# B&R Automation Studio project Panasonic_LinkaPowerCP2_A2021055 (part 18)

#### Main.st - Init, cyclic, exit code
```iecst
PROGRAM _INIT
	(* Insert code here *)

END_PROGRAM

PROGRAM _CYCLIC

    //Volanie funkcie SequenceControl//
	SequenceControl(SC:= SC_P2_StoperMaticovacky);

	//Volanie podprogramov//
	OvlCentrovacky;
	IOLinkKomunikacia;
	AtlasCopcoKomunikacia;

	//Reset sekcie //
	IF P2_StoperMaticovacky.Reset THEN
		SC_P2_StoperMaticovacky.Step:= 0;
		P2_StoperMaticovacky.Reset:= FALSE;
	ELSIF NOT Safety.STAV.Linka_ZonaCS_AKTIVNA AND NOT P2_StoperMaticovacky.Automat THEN
		SC_P2_StoperMaticovacky.Step:= 0;
	ELSIF NOT Safety.STAV.Linka_ZonaCS_AKTIVNA AND P2_StoperMaticovacky.Automat THEN
		P2_Pracovisko.STAV.Porucha_ST2:= TRUE;
	END_IF

	//Zrušenie podania matice//
	IF P2_StoperMaticovacky.SkrutSet_MaticaM4.CMD.PodajMaticu AND P2_StoperMaticovacky.SkrutSet_MaticaM4.STAV.MaticaPripravena THEN
		P2_StoperMaticovacky.SkrutSet_MaticaM4.CMD.PodajMaticu:= FALSE;
	ELSIF P2_StoperMaticovacky.SkrutSet_MaticaM4.CMD.PodajMaticu AND P2_StoperMaticovacky.SkrutSet_MaticaM4.STAV.ERROR THEN
		P2_StoperMaticovacky.SkrutSet_MaticaM4.CMD.PodajMaticu:= FALSE;
		P2_Alarmy[298]:= TRUE;
		P2_Pracovisko.STAV.Porucha_ST2:= TRUE;
	END_IF

	//Ukončenie komunikácie pri poruche//
	IF P2_Pracovisko.STAV.Porucha_ST2 AND NOT Triger_0 THEN
		Triger_0:= TRUE;
		IF P2_StoperMaticovacky.STAV.VyrobaZacala THEN
			Paletka[i].PAR.StavPowerCP:= 'FAIL';
			Paletka[i].STAV.StavPaletky:= 'NG';
			P2_StoperMaticovacky.KoniecCyklu:= TRUE;
			SC_P2_StoperMaticovacky.ResetStep:= TRUE;
			SC_P2_StoperMaticovacky.Step:= 550;
		ELSE
			SC_P2_StoperMaticovacky.ResetStep:= TRUE;
			SC_P2_StoperMaticovacky.Step:= 0;
		END_IF
	END_IF

	IF NOT P2_Pracovisko.STAV.Porucha_ST2 THEN
		Triger_0:= FALSE;
	END_IF

	CASE SC_P2_StoperMaticovacky.Step OF

		0:
			SC_P2_StoperMaticovacky.StepName:='0 - Nulovanie';
			SC_OvlCentrovacky.Step:= 0;
			P2_StoperMaticovacky.Automat:= FALSE;
			P2_StoperMaticovacky.KoniecCyklu:= FALSE;
			P2_StoperMaticovacky.Manual:= FALSE;
			P2_StoperMaticovacky.STAV.PoINIT:= FALSE;
			P2_StoperMaticovacky.STAV.VyrobaZacala:= FALSE;
			P2_StoperMaticovacky.STAV.VstupnaKamerovaKontrola:= FALSE;
			P2_StoperMaticovacky.OUT.ZasunStoper:= FALSE;
			P2_StoperMaticovacky.OUT.Maticovacku_M4_VYSUN:= FALSE;
			P2_StoperMaticovacky.OUT.Maticovacka_M4_Odvzdusn_ON:= FALSE;
			P2_StoperMaticovacky.OUT.Maticovacka_M4_Prisavanie_ON:= FALSE;
			P2_StoperMaticovacky.RFID_hlava.PrecitajChipRFID:= FALSE;
			P2_StoperMaticovacky.SkrutSet_MaticaM4.CMD.ENABLE:= FALSE;

			P2_StoperMaticovacky.Maticovacka_M4.RESET_Poruchy:= FALSE;
			P2_StoperMaticovacky.Maticovacka_M4.RESET_Vysledkov:= FALSE;
			P2_StoperMaticovacky.Maticovacka_M4.START_Skrutkovania:= FALSE;
			P2_StoperMaticovacky.Maticovacka_M4.START_Utahovania:= FALSE;
			P2_StoperMaticovacky.CMD.RR_VysunCentrovanie:= FALSE;

			CAM9.CMD.Triger:= FALSE;
			CAM9.STAV.Results_READY:= FALSE;
			FTP_CAM9.CMD.OdosliFotku:= FALSE;
			FTP_CAM9.CMD.VymazFotku:= FALSE;
			TRCB_P2_Maticovacka_ST4.CMD.VyziadajStavPaletky_TYP1:= FALSE;
			TRCB_P2_Maticovacka_ST4.CMD.PriradQRkodFiltra_TYP3:= FALSE;
			TRCB_P2_Maticovacka_ST4.CMD.OdosliStavPaletky_TYP2:= FALSE;
			TRCB_P2_Maticovacka_ST4.CMD.VyziadajStavPanatrace_TYP4:= FALSE;

			P2_StoperMaticovacky.STAV.PrebiehaVyvezeniePaletky:= FALSE;
			P2_StoperZaklTesnenia.STAV.PrebiehaVyvezeniePaletky:= FALSE;
			P2_Maticov_KAM_Result_Ignoruj:= FALSE;
			TestovaciKus:= FALSE;
			CisloFotky:= 0;
			P2_Maticov_KAM_Result_OK:= FALSE;
			P2_Maticov_KAM_Result_NG:= FALSE;
			P2_Vizu.ZobrazHL1_ST4:= FALSE;
			P2_Vizu.ZobrazHL2_ST4:= FALSE;
			P2_Vizu.ZobrazHL3_ST4:= FALSE;
			P2_Vizu.ZobrazHL4_ST4:= FALSE;
			TRCB_P2_Maticov_OpatovnyDopyt:= FALSE;
			TRCB_P2_Maticov_PaletkaNG:= FALSE;
			VysunutieSkrutkovacky_OK:= FALSE;
			PocetTrigrovKamery:= 0;
			PocetDopytovNaServer:= 0;
			CasSrobovania:= 0;
			P2_Maticovacka_Taktime.IN.START_MeraniaCasu:= FALSE;
			P2_Maticovacka_Taktime.IN.START_MeraniaStratovehoCasu:= FALSE;

			IF Safety.STAV.Linka_ZonaCS_AKTIVNA AND
				Safety.STAV.P2_ZonaBunky_AKTIVNA AND
				P2_Pracovisko.STAV.HardwareBunky_OK AND
				NOT P2_Pracovisko.STAV.Porucha_ST2 AND
				NOT P2_Pracovisko.STAV.Porucha_ST3 AND
				NOT P2_Pracovisko.STAV.Porucha_ST4 AND
				NOT P2_Pracovisko.STAV.Porucha_ST5 THEN
				SC_P2_StoperMaticovacky.ResetStep:= TRUE;
				SC_P2_StoperMaticovacky.Step:= 1;
			END_IF

		1:
			SC_P2_StoperMaticovacky.StepName:='1 - Cakam na spustenie vyroby';
			P2_StoperMaticovacky.KoniecCyklu:= FALSE;
			IF P2_StoperMaticovacky.Automat THEN
				SC_P2_StoperMaticovacky.Step:= 2;
			ELSIF P2_StoperMaticovacky.Manual THEN
				SC_P2_StoperMaticovacky.Step:= 700;
			END_IF

			//********************************************************Inicializácia****************************************************************************//

		2:
			SC_P2_StoperMaticovacky.StepName:='2 - Inicializacia - cakam na spustenie inicializacie';
			SC_P2_StoperMaticovacky.IdleTime.PT:= T#4s;
			SC_P2_StoperMaticovacky.AlarmTime.PT:= T#5s;

			P2_StoperMaticovacky.OUT.Maticovacku_M4_VYSUN:= FALSE;

			IF P2_StoperMaticovacky.IN.Maticovacka_M4_ZASUNUTA AND P2_Dopravniky.STAV.PoINIT THEN
				P2_StoperMaticovacky.SkrutSet_MaticaM4.CMD.ENABLE:= TRUE;
				SC_P2_StoperMaticovacky.ResetStep:= TRUE;
				SC_P2_StoperMaticovacky.Step:= 10;
			END_IF

		3:
			SC_P2_StoperMaticovacky.StepName:='3 - Inicializacia - vymazanie adresara kamery';
			SC_P2_StoperMaticovacky.IdleTime.PT:= T#4s;
			SC_P2_StoperMaticovacky.AlarmTime.PT:= T#5s;

			IF NOT SC_P2_StoperMaticovacky.Switch1 THEN
				FTP_CAM9.CMD.VymazFotku:= TRUE;
				SC_P2_StoperMaticovacky.Switch1:= TRUE;
			END_IF

			IF FTP_CAM9.STATUS.KomunikaciaUkoncena THEN
				FTP_CAM9.CMD.VymazFotku:= FALSE;
				SC_P2_StoperMaticovacky.ResetStep:= TRUE;
				SC_P2_StoperMaticovacky.Step:= 10;
			ELSIF FTP_CAM9.STATUS.KomunikaciaError THEN
				P2_Alarmy[229]:= TRUE;
				P2_Pracovisko.STAV.Porucha_ST2:= TRUE;
			END_IF

		10:
			SC_P2_StoperMaticovacky.StepName:='10 - Inicializacia - zasunutie centrovacky';
			SC_P2_StoperMaticovacky.IdleTime.PT:= T#4s;
			SC_P2_StoperMaticovacky.AlarmTime.PT:= T#5s;

			IF NOT SC_P2_StoperMaticovacky.Switch1 THEN
				Centrovacku_ZASUN:= TRUE;
				SC_P2_StoperMaticovacky.Switch1:= TRUE;
			END_IF

			IF P2_StoperMaticovacky.IN.Centrovanie_ZASUNUTE AND P2_Dopravniky.STAV.PoINIT THEN
				SC_P2_StoperMaticovacky.ResetStep:= TRUE;
				SC_P2_StoperMaticovacky.Step:= 12;
			END_IF

		12:
			SC_P2_StoperMaticovacky.StepName:='12 - Inicializacia - kontrola matice v maticovacke';
			SC_P2_StoperMaticovacky.IdleTime.PT:= T#5s;
			SC_P2_StoperMaticovacky.AlarmTime.PT:= T#10s;

			IF NOT SC_P2_StoperMaticovacky.Switch1 AND NOT P2_StoperMaticovacky.SkrutSet_MaticaM4.STAV.MaticaPripravena THEN
				P2_StoperMaticovacky.SkrutSet_MaticaM4.CMD.PodajMaticu:= TRUE;
				SC_P2_StoperMaticovacky.Switch1:= TRUE;
			END_IF

			IF P2_StoperMaticovacky.SkrutSet_MaticaM4.STAV.MaticaPripravena THEN
				SC_P2_StoperMaticovacky.ResetStep:= TRUE;
				SC_P2_StoperMaticovacky.Step:= 13;
			END_IF

		13:
			SC_P2_StoperMaticovacky.StepName:='13 - Inicializacia - hladanie paletky';
			SC_P2_StoperMaticovacky.IdleTime.PT:= T#5s;
			SC_P2_StoperMaticovacky.AlarmTime.PT:= T#5s;
			SC_P2_StoperMaticovacky.IdleTime.IN:= TRUE;

			IF P2_StoperMaticovacky.RFID_hlava.PritomnostPaletky THEN
				SC_P2_StoperMaticovacky.ResetStep:= TRUE;
				SC_P2_StoperMaticovacky.Step:= 20;
			ELSIF SC_P2_StoperMaticovacky.IdleTime.Q THEN
				P2_StoperMaticovacky.STAV.PoINIT:= TRUE;
				SC_P2_StoperMaticovacky.ResetStep:= TRUE;
				SC_P2_StoperMaticovacky.Step:= 100;
			END_IF

		20:
			SC_P2_StoperMaticovacky.StepName:='20 - Inicializacia - precitanie cisla paletky';
			SC_P2_StoperMaticovacky.IdleTime.PT:= T#200ms;
			SC_P2_StoperMaticovacky.AlarmTime.PT:= T#5s;

			SC_P2_StoperMaticovacky.IdleTime.IN:= P2_StoperMaticovacky.RFID_hlava.PritomnostPaletky;

			IF SC_P2_StoperMaticovacky.IdleTime.Q AND NOT SC_P2_StoperMaticovacky.Switch1 THEN
				P2_StoperMaticovacky.RFID_hlava.PrecitajChipRFID:= TRUE;
				i:= 0;
				SC_P2_StoperMaticovacky.Switch1:= TRUE;
			END_IF

			IF P2_StoperMaticovacky.RFID_hlava.Stav_CitanieZapis_OK AND P2_StoperMaticovacky.RFID_hlava.PrecitaneCisloPaletky <> 0 THEN
				i:= P2_StoperMaticovacky.RFID_hlava.PrecitaneCisloPaletky;
				P2_StoperMaticovacky.PAR.CisloPaletky:= P2_StoperMaticovacky.RFID_hlava.PrecitaneCisloPaletky;
				P2_StoperMaticovacky.RFID_hlava.PrecitajChipRFID:= FALSE;
				SC_P2_StoperMaticovacky.ResetStep:= TRUE;
				SC_P2_StoperMaticovacky.Step:= 23;
			END_IF

		23:
			SC_P2_StoperMaticovacky.StepName:='23 - Inicializacia - kontrola a priradenie indexu paletky na zaklade precitanej hodnoty';
			SC_P2_StoperMaticovacky.IdleTime.PT:= T#1s;
			SC_P2_StoperMaticovacky.AlarmTime.PT:= T#5s;

			IF i<> 0 THEN
				P2_StoperMaticovacky.PAR.CisloPaletky_STRING:= USINT_TO_STRING(i);
				Paletka[i].PAR.CisloPaletky:= USINT_TO_STRING(i);
				SC_P2_StoperMaticovacky.ResetStep:= TRUE;
				SC_P2_StoperMaticovacky.Step:= 30;
			ELSE
				P2_Alarmy[211]:= TRUE;
				P2_Pracovisko.STAV.Porucha_ST2:= TRUE;
			END_IF

		30:
			SC_P2_StoperMaticovacky.StepName:='30 - Inicializacia - kontrola stavu paletky';
			SC_P2_StoperMaticovacky.IdleTime.PT:= T#200ms;
			SC_P2_StoperMaticovacky.AlarmTime.PT:= T#5s;

			IF Paletka[i].STAV.StavPaletky = '' THEN
				Paletka[i].STAV.StavPaletky:= 'NG';
				SC_P2_StoperMaticovacky.ResetStep:= TRUE;
				SC_P2_StoperMaticovacky.Step:= 560;
			ELSIF Paletka[i].STAV.StavPaletky = 'PRECH' THEN
				P2_StoperMaticovacky.STAV.PoINIT:= TRUE;
				SC_P2_StoperMaticovacky.ResetStep:= TRUE;
				SC_P2_StoperMaticovacky.Step:= 560;
			ELSIF Paletka[i].STAV.StavPaletky = 'TEST' AND Paletka[i].STAV.CisloTestovacejStanice = 'ST_4' THEN
				TestovaciKus:= TRUE;
			ELSIF Paletka[i].STAV.StavPaletky = 'TEST' AND Paletka[i].STAV.CisloTestovacejStanice <> 'ST_4' THEN
				P2_StoperMaticovacky.STAV.PoINIT:= TRUE;
				SC_P2_StoperMaticovacky.ResetStep:= TRUE;
				SC_P2_StoperMaticovacky.Step:= 560;
			ELSIF Paletka[i].STAV.StavPaletky = 'REV' AND Paletka[i].STAV.CisloRevorkovejStanice = 'ST_4' THEN
				Paletka[i].STAV.StavPaletky:= 'OK';
				SC_P2_StoperMaticovacky.ResetStep:= TRUE;
				SC_P2_StoperMaticovacky.Step:= 33;
			ELSIF Paletka[i].STAV.StavPaletky = 'REV' AND Paletka[i].STAV.CisloRevorkovejStanice <> 'ST_4' THEN
				P2_StoperMaticovacky.STAV.PoINIT:= TRUE;
				SC_P2_StoperMaticovacky.ResetStep:= TRUE;
				SC_P2_StoperMaticovacky.Step:= 560;
			ELSIF Paletka[i].STAV.StavPaletky = 'OK' THEN
				SC_P2_StoperMaticovacky.ResetStep:= TRUE;
				SC_P2_StoperMaticovacky.Step:= 33;
			ELSIF Paletka[i].STAV.StavPaletky = 'NG' THEN
				P2_StoperMaticovacky.STAV.PoINIT:= TRUE;
				SC_P2_StoperMaticovacky.ResetStep:= TRUE;
				SC_P2_StoperMaticovacky.Step:= 560;
			END_IF

		33:
			SC_P2_StoperMaticovacky.StepName:='33 - Inicializacia - rozhodnutie podla typu modelu';
			SC_P2_StoperMaticovacky.IdleTime.PT:= T#200ms;
			SC_P2_StoperMaticovacky.AlarmTime.PT:= T#5s;

			IF Linka.PAR.ZvolenyModel = '5H' THEN
				SC_P2_StoperMaticovacky.ResetStep:= TRUE;
				SC_P2_StoperMaticovacky.Step:= 35;
			ELSE
				P2_StoperMaticovacky.STAV.PoINIT:= TRUE;
				SC_P2_StoperMaticovacky.ResetStep:= TRUE;
				SC_P2_StoperMaticovacky.Step:= 560;
			END_IF

		35:
			SC_P2_StoperMaticovacky.StepName:='35 - Inicializacia - kontrola uzavretia komunikacie';
			SC_P2_StoperMaticovacky.IdleTime.PT:= T#200ms;
			SC_P2_StoperMaticovacky.AlarmTime.PT:= T#5s;

			IF Paletka[i].STAV.Komunikacia_DONE THEN
				P2_StoperMaticovacky.STAV.PoINIT:= TRUE;
				SC_P2_StoperMaticovacky.ResetStep:= TRUE;
				SC_P2_StoperMaticovacky.Step:= 560;
			ELSE
				P2_StoperMaticovacky.STAV.PoINIT:= TRUE;
				P2_StoperMaticovacky.STAV.VstupnaKamerovaKontrola:= TRUE;
				SC_P2_StoperMaticovacky.ResetStep:= TRUE;
				SC_P2_StoperMaticovacky.Step:= 100;
			END_IF

			//********************************************************Automatický režim****************************************************************************//

		100:
			SC_P2_StoperMaticovacky.StepName:='100 - Automaticky Rezim - cakam na príchod paletky na stoper';
			SC_P2_StoperMaticovacky.IdleTime.PT:= T#200ms;
			SC_P2_StoperMaticovacky.AlarmTime.PT:= T#5s;

			SC_P2_StoperMaticovacky.IdleTime.IN:= P2_StoperMaticovacky.RFID_hlava.PritomnostPaletky;

			IF P2_StoperMaticovacky.RFID_hlava.PritomnostPaletky THEN
				P2_StoperZaklTesnenia.STAV.PrebiehaVyvezeniePaletky:= FALSE;
			END_IF

			IF NOT SC_P2_StoperMaticovacky.Switch1 AND P2_StoperMaticovacky.RFID_hlava.PritomnostPaletky THEN
				P2_Maticovacka_Taktime.IN.START_MeraniaCasu:= TRUE;
				P2_Maticovacka_Taktime.IN.ZAPIS_MeraniaCasu:= TRUE;
				P2_Maticovacka_Taktime.IN.ZAPIS_StratovyCas:= TRUE;
				Buffer_4.Hodnota:= P2_Maticovacka_Taktime.OUT.StratoveSekundy;
				Buffer_4.ZapisHodnotu:= TRUE;
				SC_P2_StoperMaticovacky.Switch1:= TRUE;
			END_IF

			IF P2_StoperMaticovacky.KoniecCyklu THEN
				SC_P2_StoperMaticovacky.ResetStep:= TRUE;
				SC_P2_StoperMaticovacky.Step:= 0;
			ELSIF SC_P2_StoperMaticovacky.IdleTime.Q THEN
				SC_P2_StoperMaticovacky.ResetStep:= TRUE;
				SC_P2_StoperMaticovacky.Step:= 101;
			END_IF

		101:
			SC_P2_StoperMaticovacky.StepName:='101 - Automaticky Rezim - precitanie cisla paletky';
			SC_P2_StoperMaticovacky.IdleTime.PT:= T#500ms;
			SC_P2_StoperMaticovacky.AlarmTime.PT:= T#5s;
			SC_P2_StoperMaticovacky.IdleTime.IN:= TRUE;

			IF NOT SC_P2_StoperMaticovacky.Switch1 THEN
				P2_StoperMaticovacky.RFID_hlava.PrecitajChipRFID:= TRUE;
				i:= 0;
				SC_P2_StoperMaticovacky.Switch1:= TRUE;
			END_IF

			IF P2_StoperMaticovacky.RFID_hlava.Stav_CitanieZapis_OK AND P2_StoperMaticovacky.RFID_hlava.PrecitaneCisloPaletky <> 0 THEN
				i:= P2_StoperMaticovacky.RFID_hlava.PrecitaneCisloPaletky;
				P2_StoperMaticovacky.PAR.CisloPaletky:= P2_StoperMaticovacky.RFID_hlava.PrecitaneCisloPaletky;
				P2_StoperMaticovacky.RFID_hlava.PrecitajChipRFID:= FALSE;
				SC_P2_StoperMaticovacky.ResetStep:= TRUE;
				SC_P2_StoperMaticovacky.Step:= 102;
			END_IF

		102:
			SC_P2_StoperMaticovacky.StepName:='102 - Automaticky Rezim - kontrola a priradenie indexu paletky na zaklade precitanej hodnoty';
			SC_P2_StoperMaticovacky.IdleTime.PT:= T#1s;
			SC_P2_StoperMaticovacky.AlarmTime.PT:= T#5s;

			IF i<> 0 THEN
				P2_StoperMaticovacky.PAR.CisloPaletky_STRING:= USINT_TO_STRING(i);
				Paletka[i].PAR.CisloPaletky:= USINT_TO_STRING(i);
				SC_P2_StoperMaticovacky.ResetStep:= TRUE;
				SC_P2_StoperMaticovacky.Step:= 103;
			ELSE
				P2_Alarmy[211]:= TRUE;
				P2_Pracovisko.STAV.Porucha_ST2:= TRUE;
			END_IF

		103:
			SC_P2_StoperMaticovacky.StepName:='103 - Automaticky Rezim - kontrola stavu paletky';
			SC_P2_StoperMaticovacky.IdleTime.PT:= T#200ms;
			SC_P2_StoperMaticovacky.AlarmTime.PT:= T#5s;

			IF Paletka[i].STAV.StavPaletky = '' THEN
				Paletka[i].STAV.StavPaletky:= 'NG';
				SC_P2_StoperMaticovacky.ResetStep:= TRUE;
				SC_P2_StoperMaticovacky.Step:= 560;
			ELSIF Paletka[i].STAV.StavPaletky = 'PRECH' THEN
				SC_P2_StoperMaticovacky.ResetStep:= TRUE;
				SC_P2_StoperMaticovacky.Step:= 560;
			ELSIF Paletka[i].STAV.StavPaletky = 'TEST' AND Paletka[i].STAV.CisloTestovacejStanice = 'ST_4' THEN
				TestovaciKus:= TRUE;
			ELSIF Paletka[i].STAV.StavPaletky = 'TEST' AND Paletka[i].STAV.CisloTestovacejStanice <> 'ST_4' THEN
				SC_P2_StoperMaticovacky.ResetStep:= TRUE;
				SC_P2_StoperMaticovacky.Step:= 560;
			ELSIF Paletka[i].STAV.StavPaletky = 'REV' AND Paletka[i].STAV.CisloRevorkovejStanice = 'ST_4' THEN
				Paletka[i].STAV.StavPaletky:= 'OK';
				SC_P2_StoperMaticovacky.ResetStep:= TRUE;
				SC_P2_StoperMaticovacky.Step:= 108;
			ELSIF Paletka[i].STAV.StavPaletky = 'REV' AND Paletka[i].STAV.CisloRevorkovejStanice <> 'ST_4' THEN
				SC_P2_StoperMaticovacky.ResetStep:= TRUE;
				SC_P2_StoperMaticovacky.Step:= 560;
			ELSIF Paletka[i].STAV.StavPaletky = 'OK' THEN
				SC_P2_StoperMaticovacky.ResetStep:= TRUE;
				SC_P2_StoperMaticovacky.Step:= 108;
			ELSIF Paletka[i].STAV.StavPaletky = 'NG' THEN
				SC_P2_StoperMaticovacky.ResetStep:= TRUE;
				SC_P2_StoperMaticovacky.Step:= 560;
			END_IF

		108:
			SC_P2_StoperMaticovacky.StepName:='108 - Automaticky Rezim - rozhodnutie podla typu modelu';
			SC_P2_StoperMaticovacky.IdleTime.PT:= T#200ms;
			SC_P2_StoperMaticovacky.AlarmTime.PT:= T#5s;

			IF Linka.PAR.ZvolenyModel = '5H' THEN
				SC_P2_StoperMaticovacky.ResetStep:= TRUE;
				SC_P2_StoperMaticovacky.Step:= 110;
			ELSE
				SC_P2_StoperMaticovacky.ResetStep:= TRUE;   //Paletka iba prechádza
				SC_P2_StoperMaticovacky.Step:= 560;
			END_IF

		110:
			SC_P2_StoperMaticovacky.StepName:='110 - Automaticky Rezim - vyziadanie stavu komunikacie zo serverom';
			SC_P2_StoperMaticovacky.IdleTime.PT:= T#200ms;
			SC_P2_StoperMaticovacky.AlarmTime.PT:= T#10s;

			IF Linka.KOM_Panatrace_OFF THEN
				SC_P2_StoperMaticovacky.ResetStep:= TRUE;
				SC_P2_StoperMaticovacky.Step:= 118;
			ELSIF NOT SC_P2_StoperMaticovacky.Switch1 AND TRCB_P2_Maticovacka_ST4.STATUS.KOM_READY THEN
				TRCB_P2_Maticovacka_ST4.CMD.VyziadajStavPanatrace_TYP4:= TRUE;
				(*P2_Maticovacka_Taktime.IN.START_MeraniaStratovehoCasu:= TRUE;*)
				Centrovacku_VYSUN:= TRUE;
				SC_P2_StoperMaticovacky.Switch1:= TRUE;
			END_IF

			IF TRCB_P2_Maticovacka_ST4.STATUS.KomunikaciaUkoncena THEN
				TRCB_P2_Maticovacka_ST4.CMD.VyziadajStavPanatrace_TYP4:= FALSE;
				P2_Maticovacka_Taktime.IN.START_MeraniaStratovehoCasu:= FALSE;
				SC_P2_StoperMaticovacky.ResetStep:= TRUE;
				SC_P2_StoperMaticovacky.Step:= 111;
			ELSIF TRCB_P2_Maticovacka_ST4.STATUS.KomunikaciaError THEN
				TRCB_P2_Maticovacka_ST4.CMD.VyziadajStavPanatrace_TYP4:= FALSE;
				P2_Maticovacka_Taktime.IN.START_MeraniaStratovehoCasu:= FALSE;
				SC_P2_StoperMaticovacky.ResetStep:= TRUE;
				SC_P2_StoperMaticovacky.Step:= 112;
			END_IF

		111:
			SC_P2_StoperMaticovacky.StepName:='111 - Automaticky Rezim - kontrola odpovede servera';
			SC_P2_StoperMaticovacky.IdleTime.PT:= T#200ms;
			SC_P2_StoperMaticovacky.AlarmTime.PT:= T#5s;

			IF NOT TRCB_P2_Maticovacka_ST4.STATUS.KomunikaciaUkoncena THEN
				IF TRCB_P2_Maticovacka_ST4.OUTPUTS.DruhCinnostiNaPaletke = '0;Generating' THEN
					SC_P2_StoperMaticovacky.ResetStep:= TRUE;
					SC_P2_StoperMaticovacky.Step:= 112;
				ELSIF TRCB_P2_Maticovacka_ST4.OUTPUTS.DruhCinnostiNaPaletke = '1;Request' THEN
					SC_P2_StoperMaticovacky.ResetStep:= TRUE;
					SC_P2_StoperMaticovacky.Step:= 113;
				ELSIF TRCB_P2_Maticovacka_ST4.OUTPUTS.DruhCinnostiNaPaletke = '2;Report' THEN
					SC_P2_StoperMaticovacky.ResetStep:= TRUE;
					SC_P2_StoperMaticovacky.Step:= 118;
				ELSIF TRCB_P2_Maticovacka_ST4.OUTPUTS.DruhCinnostiNaPaletke = '3;Wedding' THEN
					SC_P2_StoperMaticovacky.ResetStep:= TRUE;
					SC_P2_StoperMaticovacky.Step:= 112;
				ELSIF TRCB_P2_Maticovacka_ST4.OUTPUTS.DruhCinnostiNaPaletke = '4;Status' THEN
					SC_P2_StoperMaticovacky.ResetStep:= TRUE;
					SC_P2_StoperMaticovacky.Step:= 112;
				ELSIF TRCB_P2_Maticovacka_ST4.OUTPUTS.DruhCinnostiNaPaletke = '5;' THEN
					SC_P2_StoperMaticovacky.ResetStep:= TRUE;
					SC_P2_StoperMaticovacky.Step:= 112;
				ELSE
					SC_P2_StoperMaticovacky.ResetStep:= TRUE;
					SC_P2_StoperMaticovacky.Step:= 112;
				END_IF
			END_IF

		112:
			SC_P2_StoperMaticovacky.StepName:='112 - Automaticky Rezim - rozhodnutie obsluhy po chybe komunikacie s Panatrace';
			SC_P2_StoperMaticovacky.IdleTime.PT:= T#200ms;
			SC_P2_StoperMaticovacky.AlarmTime.PT:= T#5s;

			P2_Vizu.ZobrazHL4_ST4:= TRUE;

			IF TRCB_P2_Maticov_OpatovnyDopyt THEN
				TRCB_P2_Maticov_OpatovnyDopyt:= FALSE;
				P2_Vizu.ZobrazHL4_ST4:= FALSE;
				SC_P2_StoperMaticovacky.ResetStep:= TRUE;
				SC_P2_StoperMaticovacky.Step:= 110;
			ELSIF TRCB_P2_Maticov_PaletkaNG THEN
				TRCB_P2_Maticov_PaletkaNG:= FALSE;
				P2_Vizu.ZobrazHL4_ST4:= FALSE;
				Paletka[i].STAV.StavPaletky := 'NG';
				SC_P2_StoperMaticovacky.ResetStep:= TRUE;
				SC_P2_StoperMaticovacky.Step:= 116;
			END_IF

		113:
			SC_P2_StoperMaticovacky.StepName:='113 - Automaticky Rezim - vyziadanie stavu paletky zo servera';
			SC_P2_StoperMaticovacky.IdleTime.PT:= T#200ms;
			SC_P2_StoperMaticovacky.AlarmTime.PT:= T#10s;
			SC_P2_StoperMaticovacky.IdleTime.IN:= TRUE;

			IF NOT SC_P2_StoperMaticovacky.Switch1 AND TRCB_P2_Maticovacka_ST4.STATUS.KOM_READY THEN
				TRCB_P2_Maticovacka_ST4.CMD.VyziadajStavPaletky_TYP1:= TRUE;
				(*P2_Maticovacka_Taktime.IN.START_MeraniaStratovehoCasu:= TRUE;*)
				SC_P2_StoperMaticovacky.Switch1:= TRUE;
			END_IF

			IF TRCB_P2_Maticovacka_ST4.STATUS.KomunikaciaUkoncena THEN
				TRCB_P2_Maticovacka_ST4.CMD.VyziadajStavPaletky_TYP1:= FALSE;
				P2_Maticovacka_Taktime.IN.START_MeraniaStratovehoCasu:= FALSE;
				SC_P2_StoperMaticovacky.ResetStep:= TRUE;
				SC_P2_StoperMaticovacky.Step:= 114;
			ELSIF TRCB_P2_Maticovacka_ST4.STATUS.KomunikaciaError THEN
				TRCB_P2_Maticovacka_ST4.CMD.VyziadajStavPaletky_TYP1:= FALSE;
				P2_Maticovacka_Taktime.IN.START_MeraniaStratovehoCasu:= FALSE;
				SC_P2_StoperMaticovacky.ResetStep:= TRUE;
				SC_P2_StoperMaticovacky.Step:= 112;
			END_IF

		114:
			SC_P2_StoperMaticovacky.StepName:='114 - Automaticky Rezim - kontrola odpovede servera';
			SC_P2_StoperMaticovacky.IdleTime.PT:= T#200ms;
			SC_P2_StoperMaticovacky.AlarmTime.PT:= T#5s;

			IF NOT TRCB_P2_Maticovacka_ST4.STATUS.KomunikaciaUkoncena THEN
				IF TRCB_P2_Maticovacka_ST4.OUTPUTS.PovolenieCinnostiNaPaletke = 'OK' THEN
					IF TRCB_P2_Maticovacka_ST4.OUTPUTS.DruhCinnostiNaPaletke = 'PRD;ST4' THEN
						SC_P2_StoperMaticovacky.ResetStep:= TRUE;
						SC_P2_StoperMaticovacky.Step:= 118;
					END_IF
				ELSIF TRCB_P2_Maticovacka_ST4.OUTPUTS.PovolenieCinnostiNaPaletke = 'NG' THEN
					SC_P2_StoperMaticovacky.ResetStep:= TRUE;
					SC_P2_StoperMaticovacky.Step:= 115;
				END_IF
			END_IF

		115:
			SC_P2_StoperMaticovacky.StepName:='115 - Automaticky Rezim - rozhodnutie obsluhy po odpovedi panatrace NG';
			SC_P2_StoperMaticovacky.IdleTime.PT:= T#200ms;
			SC_P2_StoperMaticovacky.AlarmTime.PT:= T#5s;

			P2_Vizu.ZobrazHL3_ST4:= TRUE;

			IF TRCB_P2_Maticov_OpatovnyDopyt THEN
				TRCB_P2_Maticov_OpatovnyDopyt:= FALSE;
				P2_Vizu.ZobrazHL3_ST4:= FALSE;
				SC_P2_StoperMaticovacky.ResetStep:= TRUE;
				SC_P2_StoperMaticovacky.Step:= 110;
			ELSIF TRCB_P2_Maticov_PaletkaNG THEN
				TRCB_P2_Maticov_PaletkaNG:= FALSE;
				P2_Vizu.ZobrazHL3_ST4:= FALSE;
				Paletka[i].STAV.StavPaletky := 'NG';
				SC_P2_StoperMaticovacky.ResetStep:= TRUE;
				SC_P2_StoperMaticovacky.Step:= 116;
			END_IF

		116:
			SC_P2_StoperMaticovacky.StepName:='116 - Automaticky Rezim - odcentrovanie paletky po odpovedi servera NG';
			SC_P2_StoperMaticovacky.IdleTime.PT:= T#10s;
			SC_P2_StoperMaticovacky.AlarmTime.PT:= T#5s;

			IF NOT SC_P2_StoperMaticovacky.Switch1 THEN
				Centrovacku_ZASUN:= TRUE;
				SC_P2_StoperMaticovacky.Switch1:= TRUE;
			END_IF

			IF P2_StoperMaticovacky.IN.Centrovanie_ZASUNUTE THEN
				SC_P2_StoperMaticovacky.ResetStep:= TRUE;
				SC_P2_StoperMaticovacky.Step:= 560;
			END_IF

		118:
			SC_P2_StoperMaticovacky.StepName:='118 - Automaticky Rezim - zacentrovanie paletky';
			SC_P2_StoperMaticovacky.IdleTime.PT:= T#200ms;
			SC_P2_StoperMaticovacky.AlarmTime.PT:= T#5s;

			IF NOT SC_P2_StoperMaticovacky.Switch1 THEN
				Centrovacku_VYSUN:= TRUE;
				SC_P2_StoperMaticovacky.Switch1:= TRUE;
			END_IF

			IF P2_StoperMaticovacky.IN.Centrovanie_VYSUNUTE THEN
				CAM9.STAV.Results_READY:= FALSE;
				CAM9.STAV.OldRunCounter:= CAM9.STAV.RunCounter;
				SC_P2_StoperMaticovacky.ResetStep:= TRUE;
				SC_P2_StoperMaticovacky.Step:= 120;
			END_IF

		120:
			SC_P2_StoperMaticovacky.StepName:='120 - Automaticky Rezim - vstupna kamerova kontrola paletky CAM9';//CAM 9//
			SC_P2_StoperMaticovacky.IdleTime.PT:= T#5s;
			SC_P2_StoperMaticovacky.AlarmTime.PT:= T#5s;

			IF NOT SC_P2_StoperMaticovacky.Switch1 THEN
				CAM9.CMD.Triger:= TRUE;
				SC_P2_StoperMaticovacky.IdleTime.IN:= TRUE;
				SC_P2_StoperMaticovacky.Switch1:= TRUE;
			END_IF

			IF CAM9.STAV.Results_READY AND CAM9.STAV.OldRunCounter <> CAM9.STAV.RunCounter THEN
				PocetTrigrovKamery:= 0;
				CAM9.STAV.Results_READY:= FALSE;
				CAM9.STAV.OldRunCounter:= CAM9.STAV.RunCounter;
				SC_P2_StoperMaticovacky.ResetStep:= TRUE;
				SC_P2_StoperMaticovacky.Step:= 125;
			ELSIF SC_P2_StoperMaticovacky.IdleTime.Q AND PocetTrigrovKamery < 5 THEN
				PocetTrigrovKamery:= PocetTrigrovKamery + 1;
				CAM9.STAV.Results_READY:= FALSE;
				CAM9.STAV.OldRunCounter:= CAM9.STAV.RunCounter;
				CAM9.CMD.Triger:= FALSE;
				SC_P2_StoperMaticovacky.ResetStep:= TRUE;
				SC_P2_StoperMaticovacky.Step:= 123;
			ELSIF SC_P2_StoperMaticovacky.IdleTime.Q AND PocetTrigrovKamery >= 5 THEN
				P2_Alarmy[294]:= TRUE;
				P2_Pracovisko.STAV.Porucha_ST2:= TRUE;
			END_IF

		123:
			SC_P2_StoperMaticovacky.StepName:='123 - Automaticky Rezim - cakam na opatovny triger kamery CAM9';
			SC_P2_StoperMaticovacky.IdleTime.PT:= T#1s;
			SC_P2_StoperMaticovacky.AlarmTime.PT:= T#5s;

			SC_P2_StoperMaticovacky.IdleTime.IN:= TRUE;

			IF SC_P2_StoperMaticovacky.IdleTime.Q THEN
				SC_P2_StoperMaticovacky.ResetStep:= TRUE;
				SC_P2_StoperMaticovacky.Step:= 120;
			END_IF

		125:
			SC_P2_StoperMaticovacky.StepName:='125 - Automaticky Rezim - vysledok kamerovej kontroly paletky';
			SC_P2_StoperMaticovacky.IdleTime.PT:= T#200ms;
			SC_P2_StoperMaticovacky.AlarmTime.PT:= T#5s;
			SC_P2_StoperMaticovacky.IdleTime.IN:= TRUE;

			IF Linka.P2_Kamery_OFF THEN
				CAM9.CMD.Triger:= FALSE;
				CAM9.PAR.ResultFotky:= 'PASS';
				SC_P2_StoperMaticovacky.ResetStep:= TRUE;
				SC_P2_StoperMaticovacky.Step:= 128;
			ELSIF NOT CAM9.STAV.BUSY AND SC_P2_StoperMaticovacky.IdleTime.Q THEN
				CAM9.CMD.Triger:= FALSE;
				IF NOT CAM9.RESULT.PowerCP.PritomMatice THEN
					CAM9.PAR.ResultFotky:= 'PASS';
					SC_P2_StoperMaticovacky.ResetStep:= TRUE;
					SC_P2_StoperMaticovacky.Step:= 128;
				ELSE
					CAM9.PAR.ResultFotky:= 'FAIL';
					SC_P2_StoperMaticovacky.ResetStep:= TRUE;
					SC_P2_StoperMaticovacky.Step:= 128;
				END_IF
			END_IF

		128:
			SC_P2_StoperMaticovacky.StepName:='128 - Automaticky Rezim - rozhodnutie podla kamerovej kontroly paletky';
			SC_P2_StoperMaticovacky.IdleTime.PT:= T#200ms;
			SC_P2_StoperMaticovacky.AlarmTime.PT:= T#5s;

			IF CAM9.PAR.ResultFotky = 'PASS' THEN
				SC_P2_StoperMaticovacky.ResetStep:= TRUE;
				SC_P2_StoperMaticovacky.Step:= 130;
			ELSIF CAM9.PAR.ResultFotky = 'FAIL' THEN
				IF P2_StoperMaticovacky.STAV.VstupnaKamerovaKontrola THEN
					Paletka[i].PAR.StavPowerCP:= 'FAIL';
					Paletka[i].STAV.StavPaletky:= 'NG';
					SC_P2_StoperMaticovacky.ResetStep:= TRUE;
					SC_P2_StoperMaticovacky.Step:= 540;
				ELSE
					P2_Vizu.ZobrazHL1_ST4:= TRUE;
					IF P2_Maticov_KAM_Result_OK THEN
						P2_Maticov_KAM_Result_OK:= FALSE;
						P2_Vizu.ZobrazHL1_ST4:= FALSE;
						SC_P2_StoperMaticovacky.ResetStep:= TRUE;
						SC_P2_StoperMaticovacky.Step:= 130;
					ELSIF P2_Maticov_KAM_Result_NG THEN
						P2_Maticov_KAM_Result_NG:= FALSE;
						P2_Vizu.ZobrazHL1_ST4:= FALSE;
						Paletka[i].PAR.StavPowerCP:= 'FAIL';
						Paletka[i].STAV.StavPaletky:= 'NG';
						SC_P2_StoperMaticovacky.ResetStep:= TRUE;
						SC_P2_StoperMaticovacky.Step:= 540;
					END_IF
				END_IF
			END_IF

		130:
			SC_P2_StoperMaticovacky.StepName:='130 - Automaticky Rezim - vymazanie fotky CAM9';
			SC_P2_StoperMaticovacky.IdleTime.PT:= T#200ms;
			SC_P2_StoperMaticovacky.AlarmTime.PT:= T#5s;

			IF Linka.KOM_FTP_OFF THEN
				SC_P2_StoperMaticovacky.ResetStep:= TRUE;
				SC_P2_StoperMaticovacky.Step:= 132;
			ELSIF NOT SC_P2_StoperMaticovacky.Switch1 THEN
				FTP_CAM9.CMD.VymazFotku:= TRUE;
				SC_P2_StoperMaticovacky.Switch1:= TRUE;
			END_IF

			IF FTP_CAM9.STATUS.KomunikaciaUkoncena THEN
				FTP_CAM9.CMD.VymazFotku:= FALSE;
				SC_P2_StoperMaticovacky.ResetStep:= TRUE;
				SC_P2_StoperMaticovacky.Step:= 132;
			ELSIF FTP_CAM9.STATUS.KomunikaciaError THEN
				P2_Alarmy[229]:= TRUE;
				P2_Pracovisko.STAV.Porucha_ST2:= TRUE;
			END_IF

		132:
			SC_P2_StoperMaticovacky.StepName:='132 - Automaticky Rezim - vymazanie vysledkov skrutkovania matice M4';
			SC_P2_StoperMaticovacky.IdleTime.PT:= T#2s;
			SC_P2_StoperMaticovacky.AlarmTime.PT:= T#5s;

			IF NOT SC_P2_StoperMaticovacky.Switch1 THEN
				P2_StoperMaticovacky.Maticovacka_M4.RESET_Vysledkov:= TRUE;
				SC_P2_StoperMaticovacky.Switch1:= TRUE;
			END_IF

			IF NOT P2_StoperMaticovacky.Maticovacka_M4.Stav_VysledokUtahovania_NG AND NOT P2_StoperMaticovacky.Maticovacka_M4.Stav_VysledokUtahovania_OK THEN
				P2_StoperMaticovacky.Maticovacka_M4.RESET_Vysledkov:= FALSE;
				SC_P2_StoperMaticovacky.ResetStep:= TRUE;
				SC_P2_StoperMaticovacky.Step:= 133;
			END_IF

		133:
			SC_P2_StoperMaticovacky.StepName:='133 - Automaticky Rezim - kontrola matice M4 v skrutkovacke';
			SC_P2_StoperMaticovacky.IdleTime.PT:= T#5s;
			SC_P2_StoperMaticovacky.AlarmTime.PT:= T#2s;
			SC_P2_StoperMaticovacky.AlarmTime.IN:= TRUE;

			IF P2_StoperMaticovacky.SkrutSet_MaticaM4.STAV.MaticaPripravena THEN
				SC_P2_StoperMaticovacky.ResetStep:= TRUE;
				SC_P2_StoperMaticovacky.Step:= 136;
			ELSIF SC_P2_StoperMaticovacky.AlarmTime.Q THEN
				SC_P2_StoperMaticovacky.ResetStep:= TRUE;
				SC_P2_StoperMaticovacky.Step:= 135;
			END_IF

		135:
			SC_P2_StoperMaticovacky.StepName:='135 - Automaticky Rezim - nabitie matice do maticovacky';
			SC_P2_StoperMaticovacky.IdleTime.PT:= T#5s;
			SC_P2_StoperMaticovacky.AlarmTime.PT:= T#10s;

			IF NOT SC_P2_StoperMaticovacky.Switch1 THEN
				P2_StoperMaticovacky.SkrutSet_MaticaM4.CMD.PodajMaticu:= TRUE;
				SC_P2_StoperMaticovacky.Switch1:= TRUE;
			END_IF

			IF P2_StoperMaticovacky.SkrutSet_MaticaM4.STAV.MaticaPripravena THEN
				SC_P2_StoperMaticovacky.ResetStep:= TRUE;
				SC_P2_StoperMaticovacky.Step:= 133;
			END_IF

		136:
			SC_P2_StoperMaticovacky.StepName:='136 - Automaticky Rezim - kontrola stavu skrutkovacky matic M4';
			SC_P2_StoperMaticovacky.IdleTime.PT:= T#2s;
			SC_P2_StoperMaticovacky.AlarmTime.PT:= T#5s;

			IF P2_StoperMaticovacky.Maticovacka_M4.Stav_READY_to_START AND Safety.STAV.P2_ZonaMaticovacky_AKTIVNA THEN
				SC_P2_StoperMaticovacky.ResetStep:= TRUE;
				SC_P2_StoperMaticovacky.Step:= 138;
			END_IF

		138:
			SC_P2_StoperMaticovacky.StepName:='138 - Automaticky Rezim - start skrutkovania matic M4';
			SC_P2_StoperMaticovacky.IdleTime.PT:= T#2s;
			SC_P2_StoperMaticovacky.AlarmTime.PT:= T#5s;

			SC_P2_StoperMaticovacky.AlarmTime.IN:= (P2_StoperMaticovacky.PAR.Maticov_M4_AktualHodnVysunutia < 5);

			IF NOT SC_P2_StoperMaticovacky.Switch1 THEN
				P2_StoperMaticovacky.OUT.Maticovacka_M4_Prisavanie_ON:= TRUE;
				P2_StoperMaticovacky.OUT.Maticovacku_M4_VYSUN:= TRUE;
				P2_StoperMaticovacky.Maticovacka_M4.START_Utahovania:= TRUE;
				P2_StoperMaticovacky.STAV.VyrobaZacala:= TRUE;
				SC_P2_StoperMaticovacky.Switch1:= TRUE;
			END_IF

			IF NOT P2_StoperMaticovacky.Maticovacka_M4.Stav_UtahovanieUkoncene AND P2_StoperMaticovacky.PAR.Maticov_M4_AktualHodnVysunutia > 5 THEN
				SC_P2_StoperMaticovacky.ResetStep:= TRUE;
				SC_P2_StoperMaticovacky.Step:= 139;
			ELSIF SC_P2_StoperMaticovacky.AlarmTime.Q THEN
				P2_Alarmy[267]:= TRUE;
				P2_Pracovisko.STAV.Porucha_ST2:= TRUE;
			END_IF

		139:
			SC_P2_StoperMaticovacky.StepName:='139 - Automaticky Rezim - cakam na ukoncenie skrutkovania matic M4';
			SC_P2_StoperMaticovacky.IdleTime.PT:= T#30s;
			SC_P2_StoperMaticovacky.AlarmTime.PT:= T#10s;
			SC_P2_StoperMaticovacky.IdleTime.IN:= TRUE;
			SC_P2_StoperMaticovacky.AlarmTime.IN:= TRUE;

			IF P2_StoperMaticovacky.Maticovacka_M4.Stav_UtahovanieUkoncene THEN
				P2_StoperMaticovacky.Maticovacka_M4.START_Utahovania:= FALSE;
				CasSrobovania:= TIME_TO_REAL(SC_P2_StoperMaticovacky.IdleTime.ET);
				Reports.Skrutkovacky.VyskaSkrutkovania.P2_MaticaM4:= REAL_TO_STRING(P2_StoperMaticovacky.PAR.Maticov_M4_RoundHodnotaREAL);
				Reports.Skrutkovacky.CasSkrutkovania.P2_MaticaM4:= REAL_TO_STRING(CasSrobovania/1000);
				SC_P2_StoperMaticovacky.ResetStep:= TRUE;
				SC_P2_StoperMaticovacky.Step:= 140;
			ELSIF SC_P2_StoperMaticovacky.AlarmTime.Q THEN
				P2_Alarmy[267]:= TRUE;
				P2_Pracovisko.STAV.Porucha_ST2:= TRUE;
			END_IF

		140:
			SC_P2_StoperMaticovacky.StepName:='140 - Automaticky Rezim - zasunutie skrutkovacky matic M4 a vypnutie prisavania matice';
			SC_P2_StoperMaticovacky.IdleTime.PT:= T#200ms;
			SC_P2_StoperMaticovacky.AlarmTime.PT:= T#5s;

			IF NOT SC_P2_StoperMaticovacky.Switch1 THEN
				P2_StoperMaticovacky.OUT.Maticovacku_M4_VYSUN:= FALSE;
				P2_StoperMaticovacky.OUT.Maticovacka_M4_Prisavanie_ON:= FALSE;
				SC_P2_StoperMaticovacky.Switch1:= TRUE;
			END_IF

			IF P2_StoperMaticovacky.IN.Maticovacka_M4_ZASUNUTA THEN
				SC_P2_StoperMaticovacky.ResetStep:= TRUE;
				SC_P2_StoperMaticovacky.Step:= 143;
			END_IF

		143:
			SC_P2_StoperMaticovacky.StepName:='143 - Automaticky Rezim - nabitie matice do maticovacky';
			SC_P2_StoperMaticovacky.IdleTime.PT:= T#500ms;
			SC_P2_StoperMaticovacky.AlarmTime.PT:= T#5s;

			IF NOT SC_P2_StoperMaticovacky.Switch1 THEN
				P2_StoperMaticovacky.SkrutSet_MaticaM4.CMD.PodajMaticu:= TRUE;
				SC_P2_StoperMaticovacky.IdleTime.IN:= TRUE;
				SC_P2_StoperMaticovacky.Switch1:= TRUE;
			END_IF

			IF SC_P2_StoperMaticovacky.IdleTime.Q THEN
				IF Linka.P2_SkrutkovanieResult_OFF THEN
					SC_P2_StoperMaticovacky.ResetStep:= TRUE;
					SC_P2_StoperMaticovacky.Step:= 148;
				ELSE
					SC_P2_StoperMaticovacky.ResetStep:= TRUE;
					SC_P2_StoperMaticovacky.Step:= 145;
				END_IF
			END_IF

		145:
			SC_P2_StoperMaticovacky.StepName:='145 - Automaticky Rezim - kontrola vysledkov skrutkovania matice M4';
			SC_P2_StoperMaticovacky.IdleTime.PT:= T#200ms;
			SC_P2_StoperMaticovacky.AlarmTime.PT:= T#5s;

			Reports.Skrutkovacky.Moment_ToleranciaMIN.P2_MaticaM4:= REAL_TO_STRING(P2_StoperMaticovacky.STAV.Moment_ToleranciaMIN_REAL);
			Reports.Skrutkovacky.Moment_ToleranciaMAX.P2_MaticaM4:= REAL_TO_STRING(P2_StoperMaticovacky.STAV.Moment_ToleranciaMAX_REAL);
			Reports.Skrutkovacky.Moment_NameranaHodnota.P2_MaticaM4:= REAL_TO_STRING(P2_StoperMaticovacky.STAV.DosiahnutyMoment_REAL);
			Reports.Skrutkovacky.Uhol_ToleranciaMIN.P2_MaticaM4:= UDINT_TO_STRING(P2_StoperMaticovacky.STAV.Uhol_ToleranciaMIN);
			Reports.Skrutkovacky.Uhol_ToleranciaMAX.P2_MaticaM4:= UDINT_TO_STRING(P2_StoperMaticovacky.STAV.Uhol_ToleranciaMAX);
			Reports.Skrutkovacky.Uhol_NameranaHodnota.P2_MaticaM4:= UDINT_TO_STRING(P2_StoperMaticovacky.STAV.DosiahnutyUhol);

			IF NOT SC_P2_StoperMaticovacky.Switch1 THEN
				P2_Maticovacka_5H_Vysunutie:= STRING_TO_REAL(Reports.Skrutkovacky.VyskaSkrutkovania.P2_MaticaM4);
				IF (P2_Maticovacka_5H_Vysunutie <= P2_RemPremenne.P2_Maticovacka_Vysunutie_HI) AND (P2_Maticovacka_5H_Vysunutie >= P2_RemPremenne.P2_Maticovacka_Vysunutie_LO)THEN
					VysunutieSkrutkovacky_OK:= TRUE;
				ELSE
					VysunutieSkrutkovacky_OK:= FALSE;
				END_IF
				SC_P2_StoperMaticovacky.Switch1:= TRUE;
			END_IF

			IF P2_StoperMaticovacky.Maticovacka_M4.Stav_VysledokUtahovania_OK THEN
				IF VysunutieSkrutkovacky_OK THEN
					Reports.Skrutkovacky.VyslednyReport.P2_MaticaM4:= 'PASS';
					CAM9.STAV.Results_READY:= FALSE;
					SC_P2_StoperMaticovacky.ResetStep:= TRUE;
					SC_P2_StoperMaticovacky.Step:= 148;
				ELSE
					Paletka[i].STAV.StavPaletky:= 'NG';
					Reports.Skrutkovacky.VyslednyReport.P2_MaticaM4:= 'FAIL';
					IF P2_Maticov_MaticaM4_Result_OFF THEN
						CAM9.STAV.Results_READY:= FALSE;
						SC_P2_StoperMaticovacky.ResetStep:= TRUE;
						SC_P2_StoperMaticovacky.Step:= 148;
					ELSE
						CAM9.STAV.Results_READY:= FALSE;
						Paletka[i].PAR.StavPowerCP:= 'FAIL';
						Paletka[i].STAV.StavPaletky:= 'NG';
						SC_P2_StoperMaticovacky.ResetStep:= TRUE;
						SC_P2_StoperMaticovacky.Step:= 545;
					END_IF
				END_IF
			ELSIF P2_StoperMaticovacky.Maticovacka_M4.Stav_VysledokUtahovania_NG THEN
				Paletka[i].STAV.StavPaletky:= 'NG';
				Reports.Skrutkovacky.VyslednyReport.P2_MaticaM4:= 'FAIL';
				IF P2_Maticov_MaticaM4_Result_OFF THEN
					CAM9.STAV.Results_READY:= FALSE;
					CAM9.STAV.OldRunCounter:= CAM9.STAV.RunCounter;
					SC_P2_StoperMaticovacky.ResetStep:= TRUE;
					SC_P2_StoperMaticovacky.Step:= 148;
				ELSE
					CAM9.STAV.Results_READY:= FALSE;
					Paletka[i].PAR.StavPowerCP:= 'FAIL';
					SC_P2_StoperMaticovacky.ResetStep:= TRUE;
					SC_P2_StoperMaticovacky.Step:= 545;
				END_IF
			END_IF

		148:
			SC_P2_StoperMaticovacky.StepName:='148 - Automaticky Rezim - kamerova kontrola paletky CAM9'; //CAM 9//
			SC_P2_StoperMaticovacky.IdleTime.PT:= T#5s;
			SC_P2_StoperMaticovacky.AlarmTime.PT:= T#5s;

			IF NOT SC_P2_StoperMaticovacky.Switch1 THEN
				CAM9.CMD.Triger:= TRUE;
				SC_P2_StoperMaticovacky.IdleTime.IN:= TRUE;
				SC_P2_StoperMaticovacky.Switch1:= TRUE;
			END_IF

			IF CAM9.STAV.Results_READY AND CAM9.STAV.OldRunCounter <> CAM9.STAV.RunCounter THEN
				PocetTrigrovKamery:= 0;
				CAM9.STAV.Results_READY:= FALSE;
				CAM9.STAV.OldRunCounter:= CAM9.STAV.RunCounter;
				SC_P2_StoperMaticovacky.ResetStep:= TRUE;
				SC_P2_StoperMaticovacky.Step:= 153;
			ELSIF SC_P2_StoperMaticovacky.IdleTime.Q AND PocetTrigrovKamery < 5 THEN
				PocetTrigrovKamery:= PocetTrigrovKamery + 1;
				CAM9.STAV.Results_READY:= FALSE;
				CAM9.STAV.OldRunCounter:= CAM9.STAV.RunCounter;
				CAM9.CMD.Triger:= FALSE;
				SC_P2_StoperMaticovacky.ResetStep:= TRUE;
				SC_P2_StoperMaticovacky.Step:= 150;
			ELSIF SC_P2_StoperMaticovacky.IdleTime.Q AND PocetTrigrovKamery >= 5 THEN
				P2_Alarmy[294]:= TRUE;
				P2_Pracovisko.STAV.Porucha_ST2:= TRUE;
			END_IF

		150:
			SC_P2_StoperMaticovacky.StepName:='150 - Automaticky Rezim - cakam na opatovny triger kamery CAM9';
			SC_P2_StoperMaticovacky.IdleTime.PT:= T#1s;
			SC_P2_StoperMaticovacky.AlarmTime.PT:= T#5s;

			SC_P2_StoperMaticovacky.IdleTime.IN:= TRUE;

			IF SC_P2_StoperMaticovacky.IdleTime.Q THEN
				SC_P2_StoperMaticovacky.ResetStep:= TRUE;
				SC_P2_StoperMaticovacky.Step:= 148;
			END_IF

		153:
			SC_P2_StoperMaticovacky.StepName:='153 - Automaticky Rezim - vysledok kamerovej kontroly paletky';
			SC_P2_StoperMaticovacky.IdleTime.PT:= T#200ms;
			SC_P2_StoperMaticovacky.AlarmTime.PT:= T#5s;
			SC_P2_StoperMaticovacky.IdleTime.IN:= TRUE;

			IF Linka.P2_Kamery_OFF THEN
				CAM9.CMD.Triger:= FALSE;
				CAM9.PAR.ResultFotky:= 'PASS';
				SC_P2_StoperMaticovacky.ResetStep:= TRUE;
				SC_P2_StoperMaticovacky.Step:= 155;
			ELSIF NOT CAM9.STAV.BUSY AND SC_P2_StoperMaticovacky.IdleTime.Q THEN
				CAM9.CMD.Triger:= FALSE;
				IF CAM9.RESULT.PowerCP.PritomMatice THEN
					CAM9.PAR.ResultFotky:= 'PASS';
					SC_P2_StoperMaticovacky.ResetStep:= TRUE;
					SC_P2_StoperMaticovacky.Step:= 155;
				ELSE
					CAM9.PAR.ResultFotky:= 'FAIL';
					SC_P2_StoperMaticovacky.ResetStep:= TRUE;
					SC_P2_StoperMaticovacky.Step:= 155;
				END_IF
			END_IF

		155:
			SC_P2_StoperMaticovacky.StepName:='155 - Automaticky Rezim - rozhodnutie podla kamerovej kontroly paletky';
			SC_P2_StoperMaticovacky.IdleTime.PT:= T#200ms;
			SC_P2_StoperMaticovacky.AlarmTime.PT:= T#5s;

			IF CAM9.PAR.ResultFotky = 'PASS' THEN
				Paletka[i].PAR.StavPowerCP:= 'PASS';
				SC_P2_StoperMaticovacky.ResetStep:= TRUE;
				SC_P2_StoperMaticovacky.Step:= 540;
			ELSIF CAM9.PAR.ResultFotky = 'FAIL' THEN
				P2_Vizu.ZobrazHL2_ST4:= TRUE;
				IF P2_Maticov_KAM_Result_OK THEN
					P2_Maticov_KAM_Result_OK:= FALSE;
					P2_Vizu.ZobrazHL2_ST4:= FALSE;
					CAM9.PAR.ResultFotky:= 'PASS';
					Paletka[i].PAR.StavPowerCP:= 'PASS';
					SC_P2_StoperMaticovacky.ResetStep:= TRUE;
					SC_P2_StoperMaticovacky.Step:= 540;
				ELSIF P2_Maticov_KAM_Result_NG THEN
					P2_Maticov_KAM_Result_NG:= FALSE;
					P2_Vizu.ZobrazHL2_ST4:= FALSE;
					Paletka[i].PAR.StavPowerCP:= 'FAIL';
					Paletka[i].STAV.StavPaletky:= 'NG';
					SC_P2_StoperMaticovacky.ResetStep:= TRUE;
					SC_P2_StoperMaticovacky.Step:= 540;
				END_IF
			END_IF

			//*********************************Odoslanie fotiek na server******************************//

		540:
			SC_P2_StoperMaticovacky.StepName:='540 - Automaticky Rezim - odoslanie fotiek na server';
			SC_P2_StoperMaticovacky.IdleTime.PT:= T#200ms;
			SC_P2_StoperMaticovacky.AlarmTime.PT:= T#5s;

			IF Linka.KOM_FTP_OFF THEN
				SC_P2_StoperMaticovacky.ResetStep:= TRUE;
				SC_P2_StoperMaticovacky.Step:= 545;
			ELSIF NOT SC_P2_StoperMaticovacky.Switch1 THEN
				FTP_CAM9.INPUTS.QRkodPowerCP:= Paletka[i].PAR.QRkodPowerCP;
				CisloFotky:= CisloFotky + 1;
				FTP_CAM9.INPUTS.IndexFotky:= USINT_TO_STRING(CisloFotky);
				FTP_CAM9.INPUTS.Result:= CAM9.PAR.ResultFotky;
				Reports.Kamery.P2_CAM9_KontrolaPaletky:= CAM9.PAR.ResultFotky;
				FTP_CAM9.CMD.OdosliFotku:= TRUE;
				P2_Maticovacka_Taktime.IN.START_MeraniaStratovehoCasu:= TRUE;
				SC_P2_StoperMaticovacky.Switch1:= TRUE;
			END_IF

			IF FTP_CAM9.STATUS.KomunikaciaUkoncena THEN
				FTP_CAM9.CMD.OdosliFotku:= FALSE;
				P2_Maticovacka_Taktime.IN.START_MeraniaStratovehoCasu:= FALSE;
				Paletka[i].STAV.OdoslanieFotiek_DONE:= TRUE;
				SC_P2_StoperMaticovacky.ResetStep:= TRUE;
				SC_P2_StoperMaticovacky.Step:= 545;
			ELSIF FTP_CAM9.STATUS.KomunikaciaError THEN
				P2_Alarmy[229]:= TRUE;
				P2_Pracovisko.STAV.Porucha_ST2:= TRUE;
			END_IF

			//*********************************Odcentrovanie paletky*****************************************//

		545:
			SC_P2_StoperMaticovacky.StepName:='545 - Automaticky Rezim - odcentrovanie paletky';
			SC_P2_StoperMaticovacky.IdleTime.PT:= T#200ms;
			SC_P2_StoperMaticovacky.AlarmTime.PT:= T#5s;

			IF NOT SC_P2_StoperMaticovacky.Switch1 THEN
				Centrovacku_ZASUN:= TRUE;
				SC_P2_StoperMaticovacky.Switch1:= TRUE;
			END_IF

			IF P2_StoperMaticovacky.IN.Centrovanie_ZASUNUTE THEN
				SC_P2_StoperMaticovacky.ResetStep:= TRUE;
				SC_P2_StoperMaticovacky.Step:= 550;
			END_IF

			//*************************************Odoslanie dát na server*******************************************//

		550:
			SC_P2_StoperMaticovacky.StepName:='550 - Automaticky Rezim - odoslanie stavu paletky na server';
			SC_P2_StoperMaticovacky.IdleTime.PT:= T#200ms;
			SC_P2_StoperMaticovacky.AlarmTime.PT:= T#10s;

			IF Linka.KOM_Panatrace_OFF THEN
				SC_P2_StoperMaticovacky.ResetStep:= TRUE;
				SC_P2_StoperMaticovacky.Step:= 560;
			ELSIF NOT SC_P2_StoperMaticovacky.Switch1 AND TRCB_P2_Maticovacka_ST4.STATUS.KOM_READY THEN
				TRCB_P2_Maticovacka_ST4.CMD.OdosliStavPaletky_TYP2:= TRUE;
				(*P2_Maticovacka_Taktime.IN.START_MeraniaStratovehoCasu:= TRUE;*)
				SC_P2_StoperMaticovacky.Switch1:= TRUE;
			END_IF

			IF TRCB_P2_Maticovacka_ST4.STATUS.KomunikaciaUkoncena THEN
				TRCB_P2_Maticovacka_ST4.CMD.OdosliStavPaletky_TYP2:= FALSE;
				P2_Maticovacka_Taktime.IN.START_MeraniaStratovehoCasu:= FALSE;
				SC_P2_StoperMaticovacky.ResetStep:= TRUE;
				SC_P2_StoperMaticovacky.Step:= 552;
			ELSIF TRCB_P2_Maticovacka_ST4.STATUS.KomunikaciaError THEN
				TRCB_P2_Maticovacka_ST4.CMD.OdosliStavPaletky_TYP2:= FALSE;
				P2_Maticovacka_Taktime.IN.START_MeraniaStratovehoCasu:= FALSE;
				SC_P2_StoperMaticovacky.ResetStep:= TRUE;
				SC_P2_StoperMaticovacky.Step:= 557;
			END_IF

		552:
			SC_P2_StoperMaticovacky.StepName:='552 - Automaticky Rezim - kontrola odpovede servera';
			SC_P2_StoperMaticovacky.IdleTime.PT:= T#200ms;
			SC_P2_StoperMaticovacky.AlarmTime.PT:= T#10s;

			IF NOT TRCB_P2_Maticovacka_ST4.STATUS.KomunikaciaUkoncena THEN
				IF TRCB_P2_Maticovacka_ST4.OUTPUTS.PovolenieCinnostiNaPaletke = 'OK' THEN
					Paletka[i].STAV.Komunikacia_DONE:= TRUE;
					P2_StoperMaticovacky.STAV.VyrobaZacala:= FALSE;
					SC_P2_StoperMaticovacky.ResetStep:= TRUE;
					SC_P2_StoperMaticovacky.Step:= 560;
				ELSIF TRCB_P2_Maticovacka_ST4.OUTPUTS.PovolenieCinnostiNaPaletke = 'NG' THEN
					Paletka[i].STAV.StavPaletky:= 'NG';
					P2_StoperMaticovacky.STAV.VyrobaZacala:= FALSE;
					SC_P2_StoperMaticovacky.ResetStep:= TRUE;
					SC_P2_StoperMaticovacky.Step:= 560;
				END_IF
			END_IF

		555:
			SC_P2_StoperMaticovacky.StepName:='555 - Automaticky Rezim - vyziadanie stavu komunikacie zo serverom';
			SC_P2_StoperMaticovacky.IdleTime.PT:= T#200ms;
			SC_P2_StoperMaticovacky.AlarmTime.PT:= T#10s;

			IF NOT SC_P2_StoperMaticovacky.Switch1 AND TRCB_P2_Maticovacka_ST4.STATUS.KOM_READY THEN
				TRCB_P2_Maticovacka_ST4.CMD.VyziadajStavPanatrace_TYP4:= TRUE;
				SC_P2_StoperMaticovacky.Switch1:= TRUE;
			END_IF

			IF TRCB_P2_Maticovacka_ST4.STATUS.KomunikaciaUkoncena THEN
				TRCB_P2_Maticovacka_ST4.CMD.VyziadajStavPanatrace_TYP4:= FALSE;
				SC_P2_StoperMaticovacky.ResetStep:= TRUE;
				SC_P2_StoperMaticovacky.Step:= 556;
			ELSIF TRCB_P2_Maticovacka_ST4.STATUS.KomunikaciaError THEN
				TRCB_P2_Maticovacka_ST4.CMD.VyziadajStavPanatrace_TYP4:= FALSE;
				SC_P2_StoperMaticovacky.ResetStep:= TRUE;
				SC_P2_StoperMaticovacky.Step:= 557;
			END_IF

		556:
			SC_P2_StoperMaticovacky.StepName:='556 - Automaticky Rezim - kontrola odpovede servera';
			SC_P2_StoperMaticovacky.IdleTime.PT:= T#200ms;
			SC_P2_StoperMaticovacky.AlarmTime.PT:= T#5s;

			IF NOT TRCB_P2_Maticovacka_ST4.STATUS.KomunikaciaUkoncena THEN
				IF TRCB_P2_Maticovacka_ST4.OUTPUTS.DruhCinnostiNaPaletke = '0;Generating' THEN
					SC_P2_StoperMaticovacky.ResetStep:= TRUE;
					SC_P2_StoperMaticovacky.Step:= 557;
				ELSIF TRCB_P2_Maticovacka_ST4.OUTPUTS.DruhCinnostiNaPaletke = '1;Request' THEN
					SC_P2_StoperMaticovacky.ResetStep:= TRUE;
					SC_P2_StoperMaticovacky.Step:= 557;
				ELSIF TRCB_P2_Maticovacka_ST4.OUTPUTS.DruhCinnostiNaPaletke = '2;Report' THEN
					SC_P2_StoperMaticovacky.ResetStep:= TRUE;
					SC_P2_StoperMaticovacky.Step:= 550;
				ELSIF TRCB_P2_Maticovacka_ST4.OUTPUTS.DruhCinnostiNaPaletke = '3;Wedding' THEN
					SC_P2_StoperMaticovacky.ResetStep:= TRUE;
					SC_P2_StoperMaticovacky.Step:= 557;
				ELSIF TRCB_P2_Maticovacka_ST4.OUTPUTS.DruhCinnostiNaPaletke = '4;Status' THEN
					SC_P2_StoperMaticovacky.ResetStep:= TRUE;
					SC_P2_StoperMaticovacky.Step:= 557;
				ELSIF TRCB_P2_Maticovacka_ST4.OUTPUTS.DruhCinnostiNaPaletke = '5;' THEN
					SC_P2_StoperMaticovacky.ResetStep:= TRUE;
					SC_P2_StoperMaticovacky.Step:= 557;
				ELSE
					SC_P2_StoperMaticovacky.ResetStep:= TRUE;
					SC_P2_StoperMaticovacky.Step:= 557;
				END_IF
			END_IF

		557:
			SC_P2_StoperMaticovacky.StepName:='557 - Automaticky Rezim - rozhodnutie obsluhy po chybe komunikacie s Panatrace';
			SC_P2_StoperMaticovacky.IdleTime.PT:= T#200ms;
			SC_P2_StoperMaticovacky.AlarmTime.PT:= T#5s;

			P2_Vizu.ZobrazHL4_ST4:= TRUE;

			IF TRCB_P2_Maticov_OpatovnyDopyt THEN
				TRCB_P2_Maticov_OpatovnyDopyt:= FALSE;
				P2_Vizu.ZobrazHL4_ST4:= FALSE;
				SC_P2_StoperMaticovacky.ResetStep:= TRUE;
				SC_P2_StoperMaticovacky.Step:= 555;
			ELSIF TRCB_P2_Maticov_PaletkaNG THEN
				TRCB_P2_Maticov_PaletkaNG:= FALSE;
				P2_Vizu.ZobrazHL4_ST4:= FALSE;
				Paletka[i].STAV.StavPaletky := 'NG';
				P2_StoperMaticovacky.STAV.VyrobaZacala:= FALSE;
				SC_P2_StoperMaticovacky.ResetStep:= TRUE;
				SC_P2_StoperMaticovacky.Step:= 560;
			END_IF

			//************************************************Vyvezenie paletky******************************************************//

		560:
			SC_P2_StoperMaticovacky.StepName:='560 - Automaticky Rezim - cakam na vyvezenie na akumulacny stoper';
			SC_P2_StoperMaticovacky.IdleTime.PT:= T#200ms;
			SC_P2_StoperMaticovacky.AlarmTime.PT:= T#5s;

			IF P2_StoperMaticovacky.KoniecCyklu THEN
				SC_P2_StoperMaticovacky.ResetStep:= TRUE;
				SC_P2_StoperMaticovacky.Step:= 0;
			ELSIF P2_Pracovisko.STAV.Porucha_ST2 THEN
				SC_P2_StoperMaticovacky.ResetStep:= TRUE;
				SC_P2_StoperMaticovacky.Step:= 0;
			ELSIF ((NOT P2_AkumulacnyStoper.IN.PritomnostPaletky AND SC_P2_AkumulacnyStoper.Step = 100) OR (P2_AkumulacnyStoper.OUT.ZasunStoper AND SC_P2_AkumulacnyStoper.Step = 105)) AND NOT P2_StoperMaticovacky.STAV.PrebiehaVyvezeniePaletky THEN
				P2_StoperMaticovacky.OUT.ZasunStoper:= TRUE;
				P2_StoperMaticovacky.STAV.PrebiehaVyvezeniePaletky:= TRUE;
				SC_P2_StoperMaticovacky.ResetStep:= TRUE;
				SC_P2_StoperMaticovacky.Step:= 561;
			END_IF

		561:
			SC_P2_StoperMaticovacky.StepName:='561 - Automaticky Rezim - ukoncenie vyvazania na akumulacny stoper';
			SC_P2_StoperMaticovacky.IdleTime.PT:= T#200ms;
			SC_P2_StoperMaticovacky.AlarmTime.PT:= T#10s;

			SC_P2_StoperMaticovacky.AlarmTime.IN:= P2_StoperMaticovacky.RFID_hlava.PritomnostPaletky;
			SC_P2_StoperMaticovacky.IdleTime.IN:= NOT P2_StoperMaticovacky.RFID_hlava.PritomnostPaletky;

			IF NOT P2_StoperMaticovacky.RFID_hlava.PritomnostPaletky THEN
				TestovaciKus:= FALSE;
				CisloFotky:= 0;
				Paletka[i].PAR.StavPowerCP:= '';
				Paletka[i].STAV.Komunikacia_DONE:= FALSE;
				Paletka[i].STAV.OdoslanieFotiek_DONE:= FALSE;
				Reports.Skrutkovacky.Moment_ToleranciaMIN.P2_MaticaM4:= '';
				Reports.Skrutkovacky.Moment_ToleranciaMAX.P2_MaticaM4:= '';
				Reports.Skrutkovacky.Moment_NameranaHodnota.P2_MaticaM4:= '';
				Reports.Skrutkovacky.VyslednyReport.P2_MaticaM4:= '';
				Reports.Skrutkovacky.Uhol_ToleranciaMIN.P2_MaticaM4:= '';
				Reports.Skrutkovacky.Uhol_ToleranciaMAX.P2_MaticaM4:= '';
				Reports.Skrutkovacky.Uhol_NameranaHodnota.P2_MaticaM4:= '';
				Reports.Skrutkovacky.CasSkrutkovania.P2_MaticaM4:= '';
				Reports.Skrutkovacky.VyskaSkrutkovania.P2_MaticaM4:= '';
				Reports.Kamery.P2_CAM9_KontrolaPaletky:= '';
				P2_StoperMaticovacky.OUT.ZasunStoper:= FALSE;
				P2_StoperMaticovacky.STAV.VstupnaKamerovaKontrola:= FALSE;
				SC_P2_StoperMaticovacky.ResetStep:= TRUE;
				SC_P2_StoperMaticovacky.Step:= 100;
			ELSIF SC_P2_StoperMaticovacky.AlarmTime.Q THEN
				P2_Alarmy[287]:= TRUE;
				P2_Pracovisko.STAV.Porucha_ST2:= TRUE;
			END_IF

			//*******************************************************Manuálny režim*******************************************************************************//

		700:
			SC_P2_StoperMaticovacky.StepName:='700 - Manualny Rezim';
			SC_P2_StoperMaticovacky.IdleTime.PT:= T#8s;
			SC_P2_StoperMaticovacky.AlarmTime.PT:= T#5s;

			P2_StoperMaticovacky.SkrutSet_MaticaM4.CMD.ENABLE:= TRUE;
			P2_StoperMaticovacky.SkrutSet_MaticaM4.CMD.RucnyRezim:= TRUE;

			//Ovládanie zdvižky//
			IF P2_StoperMaticovacky.CMD.RR_VysunCentrovanie THEN
				P2_StoperMaticovacky.OUT.Centrovanie_ZASUN:= FALSE;
				P2_StoperMaticovacky.OUT.Centrovanie_VYSUN:= TRUE;
			ELSE
				P2_StoperMaticovacky.OUT.Centrovanie_ZASUN:= TRUE;
				P2_StoperMaticovacky.OUT.Centrovanie_VYSUN:= FALSE;
			END_IF

	END_CASE

END_PROGRAM

PROGRAM _EXIT
	(* Insert code here *)

END_PROGRAM
```

#### Variables.var - Local variables
```iecst
VAR
	Convert_0 : UsintToUint := (0);
	SC_OvlCentrovacky : SequenceControlTyp;
	Centrovacku_VYSUN : BOOL;
	Centrovacku_ZASUN : BOOL;
	i : USINT;
	VysunutieSkrutkovacky_OK : BOOL;
	PocetTrigrovKamery : USINT := 0;
	PocetDopytovNaServer : USINT := 0;
	TestovaciKus : BOOL := 0;
	M4_PrevodMomentu : PrevodMomentu;
	CisloFotky : USINT := 0;
	CasSrobovania : REAL := 0.0;
	P2_Maticovacka_5H_Vysunutie : REAL := 0.0;
	Triger_0 : BOOL := 0;
	Round_0 : Round;
END_VAR
```

#### IOLinkKomunikacia.st
```iecst
ACTION IOLinkKomunikacia:

	//RFID snímač paletky//
	P2_StoperMaticovacky.RFID_hlava();

	//Snímač vysunutia maticovačky M4//
	Round_0.VstupnaHodnota:= P2_StoperMaticovacky.PAR.Maticov_M4_AktualHodnVysunutia;
	P2_StoperMaticovacky.PAR.Maticov_M4_RoundHodnotaREAL:= Round_0.VystupnaHodnota;
	Round_0();

END_ACTION
```

#### OvlCentrovacky.st
```iecst
ACTION OvlCentrovacky:

	//Volanie funkcie SequenceControl//
	SequenceControl(SC:= SC_OvlCentrovacky);

	CASE SC_OvlCentrovacky.Step OF

		0:
			SC_OvlCentrovacky.StepName:= '0 - Nulovanie';
			Centrovacku_VYSUN:= FALSE;
			Centrovacku_ZASUN:= FALSE;

			IF SC_P2_StoperMaticovacky.Step <> 0 THEN
				SC_OvlCentrovacky.ResetStep:= TRUE;
				SC_OvlCentrovacky.Step:= 1;
			END_IF

		1:
			SC_OvlCentrovacky.StepName:= '1 - Rozhodnutie o cinnosti';
			IF Centrovacku_VYSUN THEN
				SC_OvlCentrovacky.Step:= 10;
			ELSIF Centrovacku_ZASUN THEN
				SC_OvlCentrovacky.Step:= 20;
			END_IF

		10:
			SC_OvlCentrovacky.StepName:= '10 - Vysunutie centrovacky';
			SC_OvlCentrovacky.IdleTime.PT:= T#3s;
			SC_OvlCentrovacky.AlarmTime.PT:= T#3s;

			IF P2_StoperMaticovacky.Automat THEN
				SC_OvlCentrovacky.AlarmTime.IN:= TRUE;
			ELSE
				SC_OvlCentrovacky.IdleTime.IN:= TRUE;
			END_IF

			IF NOT SC_OvlCentrovacky.Switch1 THEN
				P2_StoperMaticovacky.OUT.Centrovanie_ZASUN:= FALSE;
                P2_StoperMaticovacky.OUT.Centrovanie_VYSUN:= TRUE;
				SC_OvlCentrovacky.Switch1:= TRUE;
			END_IF

			IF P2_StoperMaticovacky.IN.Centrovanie_VYSUNUTE OR SC_OvlCentrovacky.IdleTime.Q THEN
				SC_OvlCentrovacky.ResetStep:= TRUE;
				SC_OvlCentrovacky.Step:= 0;
			ELSIF SC_OvlCentrovacky.AlarmTime.Q THEN
				P2_Alarmy[209]:= TRUE;
				P2_Pracovisko.STAV.Porucha_ST2:= TRUE;
			END_IF

		20:
			SC_OvlCentrovacky.StepName:= '20 - Zasunutie centrovacky';
			SC_OvlCentrovacky.IdleTime.PT:= T#3s;
			SC_OvlCentrovacky.AlarmTime.PT:= T#3s;

			IF P2_StoperMaticovacky.Automat THEN
				SC_OvlCentrovacky.AlarmTime.IN:= TRUE;
			ELSE
				SC_OvlCentrovacky.IdleTime.IN:= TRUE;
			END_IF

			IF NOT SC_OvlCentrovacky.Switch1 THEN
				P2_StoperMaticovacky.OUT.Centrovanie_VYSUN:= FALSE;
                P2_StoperMaticovacky.OUT.Centrovanie_ZASUN:= TRUE;
				SC_OvlCentrovacky.Switch1:= TRUE;
			END_IF

			IF P2_StoperMaticovacky.IN.Centrovanie_ZASUNUTE OR SC_OvlCentrovacky.IdleTime.Q THEN
				SC_OvlCentrovacky.ResetStep:= TRUE;
				SC_OvlCentrovacky.Step:= 0;
			ELSIF SC_OvlCentrovacky.AlarmTime.Q THEN
				P2_Alarmy[210]:= TRUE;
				P2_Pracovisko.STAV.Porucha_ST2:= TRUE;
			END_IF

	END_CASE

END_ACTION
```

#### AtlasCopcoKomunikacia.st
```iecst
ACTION AtlasCopcoKomunikacia:
    M4_PrevodMomentu();

	//Maticovacka M4//
	//Vstupy z AtlasCopco do PLC//
    P2_StoperMaticovacky.Maticovacka_M4.Stav_VysledokPotvrdeny:= P2_StoperMaticovacky.PAR.MaticeM4_AtlasCopcoInputs[0].0;
    P2_StoperMaticovacky.Maticovacka_M4.Stav_EmergencyStop:= P2_StoperMaticovacky.PAR.MaticeM4_AtlasCopcoInputs[0].1;
    P2_StoperMaticovacky.Maticovacka_M4.Stav_READY_to_START:= P2_StoperMaticovacky.PAR.MaticeM4_AtlasCopcoInputs[0].2;
    P2_StoperMaticovacky.Maticovacka_M4.Stav_MANUAL:= P2_StoperMaticovacky.PAR.MaticeM4_AtlasCopcoInputs[0].3;
    P2_StoperMaticovacky.Maticovacka_M4.Stav_UtahovanieUkoncene:= P2_StoperMaticovacky.PAR.MaticeM4_AtlasCopcoInputs[0].4;
    P2_StoperMaticovacky.Maticovacka_M4.Stav_VysledokUtahovania_NG:= P2_StoperMaticovacky.PAR.MaticeM4_AtlasCopcoInputs[0].5;
    P2_StoperMaticovacky.Maticovacka_M4.Stav_VysledokUtahovania_OK:= P2_StoperMaticovacky.PAR.MaticeM4_AtlasCopcoInputs[0].6;
    P2_StoperMaticovacky.Maticovacka_M4.Stav_SmerOtacania_VPRED:= P2_StoperMaticovacky.PAR.MaticeM4_AtlasCopcoInputs[0].7;
    P2_StoperMaticovacky.Maticovacka_M4.Stav_BUSY:= P2_StoperMaticovacky.PAR.MaticeM4_AtlasCopcoInputs[0].8;
    P2_StoperMaticovacky.Maticovacka_M4.Stav_ControlerSwitch_ON:= P2_StoperMaticovacky.PAR.MaticeM4_AtlasCopcoInputs[0].9;
    P2_StoperMaticovacky.Maticovacka_M4.Stav_Station_READY:= P2_StoperMaticovacky.PAR.MaticeM4_AtlasCopcoInputs[0].10;
    P2_StoperMaticovacky.Maticovacka_M4.Stav_NastrojPripojeny:= P2_StoperMaticovacky.PAR.MaticeM4_AtlasCopcoInputs[0].11;
    P2_StoperMaticovacky.Maticovacka_M4.Stav_NastrojUtahuje:= P2_StoperMaticovacky.PAR.MaticeM4_AtlasCopcoInputs[0].12;

    //Výstupy z PLC do AtlasCopco//
    P2_StoperMaticovacky.PAR.MaticeM4_AtlasCopcoOutputs[0].0:= P2_StoperMaticovacky.Maticovacka_M4.RESET_Poruchy;
    P2_StoperMaticovacky.PAR.MaticeM4_AtlasCopcoOutputs[0].1:= P2_StoperMaticovacky.Maticovacka_M4.RESET_Vysledkov;
    P2_StoperMaticovacky.PAR.MaticeM4_AtlasCopcoOutputs[0].2:= P2_StoperMaticovacky.Maticovacka_M4.START_Skrutkovania;
    P2_StoperMaticovacky.PAR.MaticeM4_AtlasCopcoOutputs[0].3:= P2_StoperMaticovacky.Maticovacka_M4.START_Utahovania;

    //Dosiahnutý moment//
//    P2_StoperMaticovacky.STAV.DosiahnutyMoment.0:= P2_StoperMaticovacky.PAR.MaticeM4_AtlasCopcoInputs[1].24;
//    P2_StoperMaticovacky.STAV.DosiahnutyMoment.1:= P2_StoperMaticovacky.PAR.MaticeM4_AtlasCopcoInputs[1].25;
//    P2_StoperMaticovacky.STAV.DosiahnutyMoment.2:= P2_StoperMaticovacky.PAR.MaticeM4_AtlasCopcoInputs[1].26;
//    P2_StoperMaticovacky.STAV.DosiahnutyMoment.3:= P2_StoperMaticovacky.PAR.MaticeM4_AtlasCopcoInputs[1].27;
//    P2_StoperMaticovacky.STAV.DosiahnutyMoment.4:= P2_StoperMaticovacky.PAR.MaticeM4_AtlasCopcoInputs[1].28;
//    P2_StoperMaticovacky.STAV.DosiahnutyMoment.5:= P2_StoperMaticovacky.PAR.MaticeM4_AtlasCopcoInputs[1].29;
//    P2_StoperMaticovacky.STAV.DosiahnutyMoment.6:= P2_StoperMaticovacky.PAR.MaticeM4_AtlasCopcoInputs[1].30;
//    P2_StoperMaticovacky.STAV.DosiahnutyMoment.7:= P2_StoperMaticovacky.PAR.MaticeM4_AtlasCopcoInputs[1].31;
//    P2_StoperMaticovacky.STAV.DosiahnutyMoment.8:= P2_StoperMaticovacky.PAR.MaticeM4_AtlasCopcoInputs[1].16;
//    P2_StoperMaticovacky.STAV.DosiahnutyMoment.9:= P2_StoperMaticovacky.PAR.MaticeM4_AtlasCopcoInputs[1].17;
//    P2_StoperMaticovacky.STAV.DosiahnutyMoment.10:= P2_StoperMaticovacky.PAR.MaticeM4_AtlasCopcoInputs[1].18;
//    P2_StoperMaticovacky.STAV.DosiahnutyMoment.11:= P2_StoperMaticovacky.PAR.MaticeM4_AtlasCopcoInputs[1].19;
//    P2_StoperMaticovacky.STAV.DosiahnutyMoment.12:= P2_StoperMaticovacky.PAR.MaticeM4_AtlasCopcoInputs[1].20;
//    P2_StoperMaticovacky.STAV.DosiahnutyMoment.13:= P2_StoperMaticovacky.PAR.MaticeM4_AtlasCopcoInputs[1].21;
//    P2_StoperMaticovacky.STAV.DosiahnutyMoment.14:= P2_StoperMaticovacky.PAR.MaticeM4_AtlasCopcoInputs[1].22;
//    P2_StoperMaticovacky.STAV.DosiahnutyMoment.15:= P2_StoperMaticovacky.PAR.MaticeM4_AtlasCopcoInputs[1].23;
//    P2_StoperMaticovacky.STAV.DosiahnutyMoment.16:= P2_StoperMaticovacky.PAR.MaticeM4_AtlasCopcoInputs[1].8;
//    P2_StoperMaticovacky.STAV.DosiahnutyMoment.17:= P2_StoperMaticovacky.PAR.MaticeM4_AtlasCopcoInputs[1].9;
//    P2_StoperMaticovacky.STAV.DosiahnutyMoment.18:= P2_StoperMaticovacky.PAR.MaticeM4_AtlasCopcoInputs[1].10;
//    P2_StoperMaticovacky.STAV.DosiahnutyMoment.19:= P2_StoperMaticovacky.PAR.MaticeM4_AtlasCopcoInputs[1].11;
//    P2_StoperMaticovacky.STAV.DosiahnutyMoment.20:= P2_StoperMaticovacky.PAR.MaticeM4_AtlasCopcoInputs[1].12;
//    P2_StoperMaticovacky.STAV.DosiahnutyMoment.21:= P2_StoperMaticovacky.PAR.MaticeM4_AtlasCopcoInputs[1].13;
//    P2_StoperMaticovacky.STAV.DosiahnutyMoment.22:= P2_StoperMaticovacky.PAR.MaticeM4_AtlasCopcoInputs[1].14;
//    P2_StoperMaticovacky.STAV.DosiahnutyMoment.23:= P2_StoperMaticovacky.PAR.MaticeM4_AtlasCopcoInputs[1].15;
//    P2_StoperMaticovacky.STAV.DosiahnutyMoment.24:= P2_StoperMaticovacky.PAR.MaticeM4_AtlasCopcoInputs[1].0;
//    P2_StoperMaticovacky.STAV.DosiahnutyMoment.25:= P2_StoperMaticovacky.PAR.MaticeM4_AtlasCopcoInputs[1].1;
//    P2_StoperMaticovacky.STAV.DosiahnutyMoment.26:= P2_StoperMaticovacky.PAR.MaticeM4_AtlasCopcoInputs[1].2;
//    P2_StoperMaticovacky.STAV.DosiahnutyMoment.27:= P2_StoperMaticovacky.PAR.MaticeM4_AtlasCopcoInputs[1].3;
//    P2_StoperMaticovacky.STAV.DosiahnutyMoment.28:= P2_StoperMaticovacky.PAR.MaticeM4_AtlasCopcoInputs[1].4;
//    P2_StoperMaticovacky.STAV.DosiahnutyMoment.29:= P2_StoperMaticovacky.PAR.MaticeM4_AtlasCopcoInputs[1].5;
//    P2_StoperMaticovacky.STAV.DosiahnutyMoment.30:= P2_StoperMaticovacky.PAR.MaticeM4_AtlasCopcoInputs[1].6;
//    P2_StoperMaticovacky.STAV.DosiahnutyMoment.31:= P2_StoperMaticovacky.PAR.MaticeM4_AtlasCopcoInputs[1].7;
//    DosiahnutyMoment_REAL:= UDINT_TO_REAL(P2_StoperMaticovacky.STAV.DosiahnutyMoment);
//    IF DosiahnutyMoment_REAL > 0 THEN
//        P2_StoperMaticovacky.STAV.DosiahnutyMoment_REAL:= DosiahnutyMoment_REAL /100;
//    ELSE
//        P2_StoperMaticovacky.STAV.DosiahnutyMoment_REAL:= 0.0;
//    END_IF

    M4_PrevodMomentu.AtlasAktualnyMoment:=P2_StoperMaticovacky.PAR.MaticeM4_AtlasCopcoInputs[1];
    P2_StoperMaticovacky.STAV.DosiahnutyMoment_REAL:=M4_PrevodMomentu.AktualnyMoment;

    //Moment - Tolerancia MAX//
//    P2_StoperMaticovacky.STAV.Moment_ToleranciaMAX.0:= P2_StoperMaticovacky.PAR.MaticeM4_AtlasCopcoInputs[3].24;
//    P2_StoperMaticovacky.STAV.Moment_ToleranciaMAX.1:= P2_StoperMaticovacky.PAR.MaticeM4_AtlasCopcoInputs[3].25;
//    P2_StoperMaticovacky.STAV.Moment_ToleranciaMAX.2:= P2_StoperMaticovacky.PAR.MaticeM4_AtlasCopcoInputs[3].26;
//    P2_StoperMaticovacky.STAV.Moment_ToleranciaMAX.3:= P2_StoperMaticovacky.PAR.MaticeM4_AtlasCopcoInputs[3].27;
//    P2_StoperMaticovacky.STAV.Moment_ToleranciaMAX.4:= P2_StoperMaticovacky.PAR.MaticeM4_AtlasCopcoInputs[3].28;
//    P2_StoperMaticovacky.STAV.Moment_ToleranciaMAX.5:= P2_StoperMaticovacky.PAR.MaticeM4_AtlasCopcoInputs[3].29;
//    P2_StoperMaticovacky.STAV.Moment_ToleranciaMAX.6:= P2_StoperMaticovacky.PAR.MaticeM4_AtlasCopcoInputs[3].30;
//    P2_StoperMaticovacky.STAV.Moment_ToleranciaMAX.7:= P2_StoperMaticovacky.PAR.MaticeM4_AtlasCopcoInputs[3].31;
//    P2_StoperMaticovacky.STAV.Moment_ToleranciaMAX.8:= P2_StoperMaticovacky.PAR.MaticeM4_AtlasCopcoInputs[3].16;
//    P2_StoperMaticovacky.STAV.Moment_ToleranciaMAX.9:= P2_StoperMaticovacky.PAR.MaticeM4_AtlasCopcoInputs[3].17;
//    P2_StoperMaticovacky.STAV.Moment_ToleranciaMAX.10:= P2_StoperMaticovacky.PAR.MaticeM4_AtlasCopcoInputs[3].18;
//    P2_StoperMaticovacky.STAV.Moment_ToleranciaMAX.11:= P2_StoperMaticovacky.PAR.MaticeM4_AtlasCopcoInputs[3].19;
//    P2_StoperMaticovacky.STAV.Moment_ToleranciaMAX.12:= P2_StoperMaticovacky.PAR.MaticeM4_AtlasCopcoInputs[3].20;
//    P2_StoperMaticovacky.STAV.Moment_ToleranciaMAX.13:= P2_StoperMaticovacky.PAR.MaticeM4_AtlasCopcoInputs[3].21;
//    P2_StoperMaticovacky.STAV.Moment_ToleranciaMAX.14:= P2_StoperMaticovacky.PAR.MaticeM4_AtlasCopcoInputs[3].22;
//    P2_StoperMaticovacky.STAV.Moment_ToleranciaMAX.15:= P2_StoperMaticovacky.PAR.MaticeM4_AtlasCopcoInputs[3].23;
//    P2_StoperMaticovacky.STAV.Moment_ToleranciaMAX.16:= P2_StoperMaticovacky.PAR.MaticeM4_AtlasCopcoInputs[3].8;
//    P2_StoperMaticovacky.STAV.Moment_ToleranciaMAX.17:= P2_StoperMaticovacky.PAR.MaticeM4_AtlasCopcoInputs[3].9;
//    P2_StoperMaticovacky.STAV.Moment_ToleranciaMAX.18:= P2_StoperMaticovacky.PAR.MaticeM4_AtlasCopcoInputs[3].10;
//    P2_StoperMaticovacky.STAV.Moment_ToleranciaMAX.19:= P2_StoperMaticovacky.PAR.MaticeM4_AtlasCopcoInputs[3].11;
//    P2_StoperMaticovacky.STAV.Moment_ToleranciaMAX.20:= P2_StoperMaticovacky.PAR.MaticeM4_AtlasCopcoInputs[3].12;
//    P2_StoperMaticovacky.STAV.Moment_ToleranciaMAX.21:= P2_StoperMaticovacky.PAR.MaticeM4_AtlasCopcoInputs[3].13;
//    P2_StoperMaticovacky.STAV.Moment_ToleranciaMAX.22:= P2_StoperMaticovacky.PAR.MaticeM4_AtlasCopcoInputs[3].14;
//    P2_StoperMaticovacky.STAV.Moment_ToleranciaMAX.23:= P2_StoperMaticovacky.PAR.MaticeM4_AtlasCopcoInputs[3].15;
//    P2_StoperMaticovacky.STAV.Moment_ToleranciaMAX.24:= P2_StoperMaticovacky.PAR.MaticeM4_AtlasCopcoInputs[3].0;
//    P2_StoperMaticovacky.STAV.Moment_ToleranciaMAX.25:= P2_StoperMaticovacky.PAR.MaticeM4_AtlasCopcoInputs[3].1;
//    P2_StoperMaticovacky.STAV.Moment_ToleranciaMAX.26:= P2_StoperMaticovacky.PAR.MaticeM4_AtlasCopcoInputs[3].2;
//    P2_StoperMaticovacky.STAV.Moment_ToleranciaMAX.27:= P2_StoperMaticovacky.PAR.MaticeM4_AtlasCopcoInputs[3].3;
//    P2_StoperMaticovacky.STAV.Moment_ToleranciaMAX.28:= P2_StoperMaticovacky.PAR.MaticeM4_AtlasCopcoInputs[3].4;
//    P2_StoperMaticovacky.STAV.Moment_ToleranciaMAX.29:= P2_StoperMaticovacky.PAR.MaticeM4_AtlasCopcoInputs[3].5;
//    P2_StoperMaticovacky.STAV.Moment_ToleranciaMAX.30:= P2_StoperMaticovacky.PAR.MaticeM4_AtlasCopcoInputs[3].6;
//    P2_StoperMaticovacky.STAV.Moment_ToleranciaMAX.31:= P2_StoperMaticovacky.PAR.MaticeM4_AtlasCopcoInputs[3].7;
//    Moment_ToleranciaMAX_REAL:= UDINT_TO_REAL(P2_StoperMaticovacky.STAV.Moment_ToleranciaMAX);
//    IF Moment_ToleranciaMAX_REAL > 0 THEN
//        P2_StoperMaticovacky.STAV.Moment_ToleranciaMAX_REAL:= Moment_ToleranciaMAX_REAL /100;
//    ELSE
//        P2_StoperMaticovacky.STAV.Moment_ToleranciaMAX_REAL:= 0.0;
//    END_IF

    M4_PrevodMomentu.AtlasMaximalnaTolerancia:=P2_StoperMaticovacky.PAR.MaticeM4_AtlasCopcoInputs[3];
    P2_StoperMaticovacky.STAV.Moment_ToleranciaMAX_REAL:=M4_PrevodMomentu.ToleranciaMAX;

    //Moment - Tolerancia MIN//
//    P2_StoperMaticovacky.STAV.Moment_ToleranciaMIN.0:= P2_StoperMaticovacky.PAR.MaticeM4_AtlasCopcoInputs[4].24;
//    P2_StoperMaticovacky.STAV.Moment_ToleranciaMIN.1:= P2_StoperMaticovacky.PAR.MaticeM4_AtlasCopcoInputs[4].25;
//    P2_StoperMaticovacky.STAV.Moment_ToleranciaMIN.2:= P2_StoperMaticovacky.PAR.MaticeM4_AtlasCopcoInputs[4].26;
//    P2_StoperMaticovacky.STAV.Moment_ToleranciaMIN.3:= P2_StoperMaticovacky.PAR.MaticeM4_AtlasCopcoInputs[4].27;
//    P2_StoperMaticovacky.STAV.Moment_ToleranciaMIN.4:= P2_StoperMaticovacky.PAR.MaticeM4_AtlasCopcoInputs[4].28;
//    P2_StoperMaticovacky.STAV.Moment_ToleranciaMIN.5:= P2_StoperMaticovacky.PAR.MaticeM4_AtlasCopcoInputs[4].29;
//    P2_StoperMaticovacky.STAV.Moment_ToleranciaMIN.6:= P2_StoperMaticovacky.PAR.MaticeM4_AtlasCopcoInputs[4].30;
//    P2_StoperMaticovacky.STAV.Moment_ToleranciaMIN.7:= P2_StoperMaticovacky.PAR.MaticeM4_AtlasCopcoInputs[4].31;
//    P2_StoperMaticovacky.STAV.Moment_ToleranciaMIN.8:= P2_StoperMaticovacky.PAR.MaticeM4_AtlasCopcoInputs[4].16;
//    P2_StoperMaticovacky.STAV.Moment_ToleranciaMIN.9:= P2_StoperMaticovacky.PAR.MaticeM4_AtlasCopcoInputs[4].17;
//    P2_StoperMaticovacky.STAV.Moment_ToleranciaMIN.10:= P2_StoperMaticovacky.PAR.MaticeM4_AtlasCopcoInputs[4].18;
//    P2_StoperMaticovacky.STAV.Moment_ToleranciaMIN.11:= P2_StoperMaticovacky.PAR.MaticeM4_AtlasCopcoInputs[4].19;
//    P2_StoperMaticovacky.STAV.Moment_ToleranciaMIN.12:= P2_StoperMaticovacky.PAR.MaticeM4_AtlasCopcoInputs[4].20;
//    P2_StoperMaticovacky.STAV.Moment_ToleranciaMIN.13:= P2_StoperMaticovacky.PAR.MaticeM4_AtlasCopcoInputs[4].21;
//    P2_StoperMaticovacky.STAV.Moment_ToleranciaMIN.14:= P2_StoperMaticovacky.PAR.MaticeM4_AtlasCopcoInputs[4].22;
//    P2_StoperMaticovacky.STAV.Moment_ToleranciaMIN.15:= P2_StoperMaticovacky.PAR.MaticeM4_AtlasCopcoInputs[4].23;
//    P2_StoperMaticovacky.STAV.Moment_ToleranciaMIN.16:= P2_StoperMaticovacky.PAR.MaticeM4_AtlasCopcoInputs[4].8;
//    P2_StoperMaticovacky.STAV.Moment_ToleranciaMIN.17:= P2_StoperMaticovacky.PAR.MaticeM4_AtlasCopcoInputs[4].9;
//    P2_StoperMaticovacky.STAV.Moment_ToleranciaMIN.18:= P2_StoperMaticovacky.PAR.MaticeM4_AtlasCopcoInputs[4].10;
//    P2_StoperMaticovacky.STAV.Moment_ToleranciaMIN.19:= P2_StoperMaticovacky.PAR.MaticeM4_AtlasCopcoInputs[4].11;
//    P2_StoperMaticovacky.STAV.Moment_ToleranciaMIN.20:= P2_StoperMaticovacky.PAR.MaticeM4_AtlasCopcoInputs[4].12;
//    P2_StoperMaticovacky.STAV.Moment_ToleranciaMIN.21:= P2_StoperMaticovacky.PAR.MaticeM4_AtlasCopcoInputs[4].13;
//    P2_StoperMaticovacky.STAV.Moment_ToleranciaMIN.22:= P2_StoperMaticovacky.PAR.MaticeM4_AtlasCopcoInputs[4].14;
//    P2_StoperMaticovacky.STAV.Moment_ToleranciaMIN.23:= P2_StoperMaticovacky.PAR.MaticeM4_AtlasCopcoInputs[4].15;
//    P2_StoperMaticovacky.STAV.Moment_ToleranciaMIN.24:= P2_StoperMaticovacky.PAR.MaticeM4_AtlasCopcoInputs[4].0;
//    P2_StoperMaticovacky.STAV.Moment_ToleranciaMIN.25:= P2_StoperMaticovacky.PAR.MaticeM4_AtlasCopcoInputs[4].1;
//    P2_StoperMaticovacky.STAV.Moment_ToleranciaMIN.26:= P2_StoperMaticovacky.PAR.MaticeM4_AtlasCopcoInputs[4].2;
//    P2_StoperMaticovacky.STAV.Moment_ToleranciaMIN.27:= P2_StoperMaticovacky.PAR.MaticeM4_AtlasCopcoInputs[4].3;
//    P2_StoperMaticovacky.STAV.Moment_ToleranciaMIN.28:= P2_StoperMaticovacky.PAR.MaticeM4_AtlasCopcoInputs[4].4;
//    P2_StoperMaticovacky.STAV.Moment_ToleranciaMIN.29:= P2_StoperMaticovacky.PAR.MaticeM4_AtlasCopcoInputs[4].5;
//    P2_StoperMaticovacky.STAV.Moment_ToleranciaMIN.30:= P2_StoperMaticovacky.PAR.MaticeM4_AtlasCopcoInputs[4].6;
//    P2_StoperMaticovacky.STAV.Moment_ToleranciaMIN.31:= P2_StoperMaticovacky.PAR.MaticeM4_AtlasCopcoInputs[4].7;
//    Moment_ToleranciaMIN_REAL:= UDINT_TO_REAL(P2_StoperMaticovacky.STAV.Moment_ToleranciaMIN);
//    IF Moment_ToleranciaMIN_REAL > 0 THEN
//        P2_StoperMaticovacky.STAV.Moment_ToleranciaMIN_REAL:= Moment_ToleranciaMIN_REAL/100;
//    ELSE
//        P2_StoperMaticovacky.STAV.Moment_ToleranciaMIN_REAL:= 0.0;
//    END_IF

    M4_PrevodMomentu.AtlasMinimalnaTolerancia:=P2_StoperMaticovacky.PAR.MaticeM4_AtlasCopcoInputs[4];
    P2_StoperMaticovacky.STAV.Moment_ToleranciaMIN_REAL:=M4_PrevodMomentu.ToleranciaMIN;

    //Dosiahnutý úhol//
    P2_StoperMaticovacky.STAV.DosiahnutyUhol.0:= P2_StoperMaticovacky.PAR.MaticeM4_AtlasCopcoInputs[0].24;
    P2_StoperMaticovacky.STAV.DosiahnutyUhol.1:= P2_StoperMaticovacky.PAR.MaticeM4_AtlasCopcoInputs[0].25;
    P2_StoperMaticovacky.STAV.DosiahnutyUhol.2:= P2_StoperMaticovacky.PAR.MaticeM4_AtlasCopcoInputs[0].26;
    P2_StoperMaticovacky.STAV.DosiahnutyUhol.3:= P2_StoperMaticovacky.PAR.MaticeM4_AtlasCopcoInputs[0].27;
    P2_StoperMaticovacky.STAV.DosiahnutyUhol.4:= P2_StoperMaticovacky.PAR.MaticeM4_AtlasCopcoInputs[0].28;
    P2_StoperMaticovacky.STAV.DosiahnutyUhol.5:= P2_StoperMaticovacky.PAR.MaticeM4_AtlasCopcoInputs[0].29;
    P2_StoperMaticovacky.STAV.DosiahnutyUhol.6:= P2_StoperMaticovacky.PAR.MaticeM4_AtlasCopcoInputs[0].30;
    P2_StoperMaticovacky.STAV.DosiahnutyUhol.7:= P2_StoperMaticovacky.PAR.MaticeM4_AtlasCopcoInputs[0].31;
    P2_StoperMaticovacky.STAV.DosiahnutyUhol.8:= P2_StoperMaticovacky.PAR.MaticeM4_AtlasCopcoInputs[0].16;
    P2_StoperMaticovacky.STAV.DosiahnutyUhol.9:= P2_StoperMaticovacky.PAR.MaticeM4_AtlasCopcoInputs[0].17;
    P2_StoperMaticovacky.STAV.DosiahnutyUhol.10:= P2_StoperMaticovacky.PAR.MaticeM4_AtlasCopcoInputs[0].18;
    P2_StoperMaticovacky.STAV.DosiahnutyUhol.11:= P2_StoperMaticovacky.PAR.MaticeM4_AtlasCopcoInputs[0].19;
    P2_StoperMaticovacky.STAV.DosiahnutyUhol.12:= P2_StoperMaticovacky.PAR.MaticeM4_AtlasCopcoInputs[0].20;
    P2_StoperMaticovacky.STAV.DosiahnutyUhol.13:= P2_StoperMaticovacky.PAR.MaticeM4_AtlasCopcoInputs[0].21;
    P2_StoperMaticovacky.STAV.DosiahnutyUhol.14:= P2_StoperMaticovacky.PAR.MaticeM4_AtlasCopcoInputs[0].22;
    P2_StoperMaticovacky.STAV.DosiahnutyUhol.15:= P2_StoperMaticovacky.PAR.MaticeM4_AtlasCopcoInputs[0].23;

    //Uhol - Tolerancia MAX//
    P2_StoperMaticovacky.STAV.Uhol_ToleranciaMAX.0:= P2_StoperMaticovacky.PAR.MaticeM4_AtlasCopcoInputs[2].8;
    P2_StoperMaticovacky.STAV.Uhol_ToleranciaMAX.1:= P2_StoperMaticovacky.PAR.MaticeM4_AtlasCopcoInputs[2].9;
    P2_StoperMaticovacky.STAV.Uhol_ToleranciaMAX.2:= P2_StoperMaticovacky.PAR.MaticeM4_AtlasCopcoInputs[2].10;
    P2_StoperMaticovacky.STAV.Uhol_ToleranciaMAX.3:= P2_StoperMaticovacky.PAR.MaticeM4_AtlasCopcoInputs[2].11;
    P2_StoperMaticovacky.STAV.Uhol_ToleranciaMAX.4:= P2_StoperMaticovacky.PAR.MaticeM4_AtlasCopcoInputs[2].12;
    P2_StoperMaticovacky.STAV.Uhol_ToleranciaMAX.5:= P2_StoperMaticovacky.PAR.MaticeM4_AtlasCopcoInputs[2].13;
    P2_StoperMaticovacky.STAV.Uhol_ToleranciaMAX.6:= P2_StoperMaticovacky.PAR.MaticeM4_AtlasCopcoInputs[2].14;
    P2_StoperMaticovacky.STAV.Uhol_ToleranciaMAX.7:= P2_StoperMaticovacky.PAR.MaticeM4_AtlasCopcoInputs[2].15;
    P2_StoperMaticovacky.STAV.Uhol_ToleranciaMAX.8:= P2_StoperMaticovacky.PAR.MaticeM4_AtlasCopcoInputs[2].0;
    P2_StoperMaticovacky.STAV.Uhol_ToleranciaMAX.9:= P2_StoperMaticovacky.PAR.MaticeM4_AtlasCopcoInputs[2].1;
    P2_StoperMaticovacky.STAV.Uhol_ToleranciaMAX.10:= P2_StoperMaticovacky.PAR.MaticeM4_AtlasCopcoInputs[2].2;
    P2_StoperMaticovacky.STAV.Uhol_ToleranciaMAX.11:= P2_StoperMaticovacky.PAR.MaticeM4_AtlasCopcoInputs[2].3;
    P2_StoperMaticovacky.STAV.Uhol_ToleranciaMAX.12:= P2_StoperMaticovacky.PAR.MaticeM4_AtlasCopcoInputs[2].4;
    P2_StoperMaticovacky.STAV.Uhol_ToleranciaMAX.13:= P2_StoperMaticovacky.PAR.MaticeM4_AtlasCopcoInputs[2].5;
    P2_StoperMaticovacky.STAV.Uhol_ToleranciaMAX.14:= P2_StoperMaticovacky.PAR.MaticeM4_AtlasCopcoInputs[2].6;
    P2_StoperMaticovacky.STAV.Uhol_ToleranciaMAX.15:= P2_StoperMaticovacky.PAR.MaticeM4_AtlasCopcoInputs[2].7;

    //Uhol - Tolerancia MIN//
    P2_StoperMaticovacky.STAV.Uhol_ToleranciaMIN.0:= P2_StoperMaticovacky.PAR.MaticeM4_AtlasCopcoInputs[2].24;
    P2_StoperMaticovacky.STAV.Uhol_ToleranciaMIN.1:= P2_StoperMaticovacky.PAR.MaticeM4_AtlasCopcoInputs[2].25;
    P2_StoperMaticovacky.STAV.Uhol_ToleranciaMIN.2:= P2_StoperMaticovacky.PAR.MaticeM4_AtlasCopcoInputs[2].26;
    P2_StoperMaticovacky.STAV.Uhol_ToleranciaMIN.3:= P2_StoperMaticovacky.PAR.MaticeM4_AtlasCopcoInputs[2].27;
    P2_StoperMaticovacky.STAV.Uhol_ToleranciaMIN.4:= P2_StoperMaticovacky.PAR.MaticeM4_AtlasCopcoInputs[2].28;
    P2_StoperMaticovacky.STAV.Uhol_ToleranciaMIN.5:= P2_StoperMaticovacky.PAR.MaticeM4_AtlasCopcoInputs[2].29;
    P2_StoperMaticovacky.STAV.Uhol_ToleranciaMIN.6:= P2_StoperMaticovacky.PAR.MaticeM4_AtlasCopcoInputs[2].30;
    P2_StoperMaticovacky.STAV.Uhol_ToleranciaMIN.7:= P2_StoperMaticovacky.PAR.MaticeM4_AtlasCopcoInputs[2].31;
    P2_StoperMaticovacky.STAV.Uhol_ToleranciaMIN.8:= P2_StoperMaticovacky.PAR.MaticeM4_AtlasCopcoInputs[2].16;
    P2_StoperMaticovacky.STAV.Uhol_ToleranciaMIN.9:= P2_StoperMaticovacky.PAR.MaticeM4_AtlasCopcoInputs[2].17;
    P2_StoperMaticovacky.STAV.Uhol_ToleranciaMIN.10:= P2_StoperMaticovacky.PAR.MaticeM4_AtlasCopcoInputs[2].18;
    P2_StoperMaticovacky.STAV.Uhol_ToleranciaMIN.11:= P2_StoperMaticovacky.PAR.MaticeM4_AtlasCopcoInputs[2].19;
    P2_StoperMaticovacky.STAV.Uhol_ToleranciaMIN.12:= P2_StoperMaticovacky.PAR.MaticeM4_AtlasCopcoInputs[2].20;
    P2_StoperMaticovacky.STAV.Uhol_ToleranciaMIN.13:= P2_StoperMaticovacky.PAR.MaticeM4_AtlasCopcoInputs[2].21;
    P2_StoperMaticovacky.STAV.Uhol_ToleranciaMIN.14:= P2_StoperMaticovacky.PAR.MaticeM4_AtlasCopcoInputs[2].22;
    P2_StoperMaticovacky.STAV.Uhol_ToleranciaMIN.15:= P2_StoperMaticovacky.PAR.MaticeM4_AtlasCopcoInputs[2].23;

END_ACTION
```

### Program Logical/Program/Pracovisko_2/P2_AkumStoper (IEC)

#### Main.st - Init, cyclic, exit code
```iecst
PROGRAM _INIT
	(* Insert code here *)

END_PROGRAM

PROGRAM _CYCLIC

	//Volanie funkcie SequenceControl//
	SequenceControl(SC:= SC_P2_AkumulacnyStoper);

	//Reset sekcie //
	IF P2_AkumulacnyStoper.Reset THEN
		SC_P2_AkumulacnyStoper.Step:= 0;
		P2_AkumulacnyStoper.Reset:= FALSE;
	ELSIF NOT Safety.STAV.Linka_ZonaCS_AKTIVNA THEN
		SC_P2_AkumulacnyStoper.Step:= 0;
	END_IF

	CASE SC_P2_AkumulacnyStoper.Step OF

		0:
			SC_P2_AkumulacnyStoper.StepName:='0 - Nulovanie';
			P2_AkumulacnyStoper.Automat:= FALSE;
			P2_AkumulacnyStoper.KoniecCyklu:= FALSE;
			P2_AkumulacnyStoper.Manual:= FALSE;
			P2_AkumulacnyStoper.STAV.PoINIT:= FALSE;
			P2_AkumulacnyStoper.STAV.PrebiehaVyvezeniePaletky:= FALSE;
			P2_StoperMaticovacky.STAV.PrebiehaVyvezeniePaletky:= FALSE;
			P2_AkumulacnyStoper.OUT.ZasunStoper:= FALSE;

			IF Safety.STAV.Linka_ZonaCS_AKTIVNA AND
				Safety.STAV.P2_ZonaBunky_AKTIVNA AND
				P2_Pracovisko.STAV.HardwareBunky_OK AND
				NOT P2_Pracovisko.STAV.Porucha_ST2 AND
				NOT P2_Pracovisko.STAV.Porucha_ST3 AND
				NOT P2_Pracovisko.STAV.Porucha_ST4 AND
				NOT P2_Pracovisko.STAV.Porucha_ST5 THEN
				SC_P2_AkumulacnyStoper.ResetStep:= TRUE;
				SC_P2_AkumulacnyStoper.Step:= 1;
			END_IF

		1:
			SC_P2_AkumulacnyStoper.StepName:='1 - Cakam na spustenie vyroby';
			P2_AkumulacnyStoper.KoniecCyklu:= FALSE;
			IF P2_AkumulacnyStoper.Automat THEN
				SC_P2_AkumulacnyStoper.Step:= 2;
			ELSIF P2_AkumulacnyStoper.Manual THEN
				SC_P2_AkumulacnyStoper.Step:= 700;
			END_IF

			//********************************************************Inicializácia****************************************************************************//
		2:
			SC_P2_AkumulacnyStoper.StepName:='2 - Inicializacia - cakam na spustenie inicializacie';
			SC_P2_AkumulacnyStoper.IdleTime.PT:= T#4s;
			SC_P2_AkumulacnyStoper.AlarmTime.PT:= T#5s;

			IF P2_Dopravniky.STAV.PoINIT THEN
				SC_P2_AkumulacnyStoper.ResetStep:= TRUE;
				SC_P2_AkumulacnyStoper.Step:= 3;
			END_IF

		3:
			SC_P2_AkumulacnyStoper.StepName:='3 - Inicializacia - hladanie paletky';
			SC_P2_AkumulacnyStoper.IdleTime.PT:= T#5s;
			SC_P2_AkumulacnyStoper.AlarmTime.PT:= T#5s;
			SC_P2_AkumulacnyStoper.IdleTime.IN:= TRUE;

			IF P2_AkumulacnyStoper.IN.PritomnostPaletky THEN
				P2_AkumulacnyStoper.STAV.PoINIT:= TRUE;
				SC_P2_AkumulacnyStoper.ResetStep:= TRUE;
				SC_P2_AkumulacnyStoper.Step:= 100;
			ELSIF SC_P2_AkumulacnyStoper.IdleTime.Q THEN
				P2_AkumulacnyStoper.STAV.PoINIT:= TRUE;
				SC_P2_AkumulacnyStoper.ResetStep:= TRUE;
				SC_P2_AkumulacnyStoper.Step:= 100;
			END_IF

			//********************************************************Automatický režim****************************************************************************//
		100:
			SC_P2_AkumulacnyStoper.StepName:='100 - Automaticky Rezim - cakam na príchod paletky na stoper';
			SC_P2_AkumulacnyStoper.IdleTime.PT:= T#200ms;
			SC_P2_AkumulacnyStoper.AlarmTime.PT:= T#5s;

			SC_P2_AkumulacnyStoper.IdleTime.IN:= P2_AkumulacnyStoper.IN.PritomnostPaletky;

			IF P2_AkumulacnyStoper.IN.PritomnostPaletky THEN
				P2_StoperMaticovacky.STAV.PrebiehaVyvezeniePaletky:= FALSE;
			END_IF

			IF P2_AkumulacnyStoper.KoniecCyklu THEN
				SC_P2_AkumulacnyStoper.ResetStep:= TRUE;
				SC_P2_AkumulacnyStoper.Step:= 0;
			ELSIF SC_P2_AkumulacnyStoper.IdleTime.Q THEN
				SC_P2_AkumulacnyStoper.ResetStep:= TRUE;
				SC_P2_AkumulacnyStoper.Step:= 101;
			END_IF

		101:
			SC_P2_AkumulacnyStoper.StepName:='101 - Automaticky Rezim - cakam na vyvezenie paletky na stoper srobovania';
			SC_P2_AkumulacnyStoper.IdleTime.PT:= T#200ms;
			SC_P2_AkumulacnyStoper.AlarmTime.PT:= T#5s;

			IF P2_AkumulacnyStoper.KoniecCyklu THEN
				SC_P2_AkumulacnyStoper.ResetStep:= TRUE;
				SC_P2_AkumulacnyStoper.Step:= 0;
			ELSIF ((NOT P2_StoperSrobovania.RFID_hlava.PritomnostPaletky AND SC_P2_StoperSrobovania.Step = 100) OR (P2_StoperSrobovania.OUT.ZasunStoper AND SC_P2_StoperSrobovania.Step = 561)) AND NOT P2_AkumulacnyStoper.STAV.PrebiehaVyvezeniePaletky AND NOT TEST THEN
				SC_P2_AkumulacnyStoper.ResetStep:= TRUE;
				SC_P2_AkumulacnyStoper.Step:= 105;
			ELSIF NOT P2_AkumulacnyStoper.IN.PritomnostPaletky THEN
				SC_P2_AkumulacnyStoper.ResetStep:= TRUE;
				SC_P2_AkumulacnyStoper.Step:= 100;
			END_IF

		105:
			SC_P2_AkumulacnyStoper.StepName:='105 - Automaticky Rezim - vyvazam paletku na stoper srobovania';
			SC_P2_AkumulacnyStoper.IdleTime.PT:= T#200ms;
			SC_P2_AkumulacnyStoper.AlarmTime.PT:= T#10s;

			SC_P2_AkumulacnyStoper.AlarmTime.IN:= P2_AkumulacnyStoper.IN.PritomnostPaletky;

			IF NOT SC_P2_AkumulacnyStoper.Switch1 THEN
				P2_AkumulacnyStoper.OUT.ZasunStoper:= TRUE;
				P2_AkumulacnyStoper.STAV.PrebiehaVyvezeniePaletky:= TRUE;
				SC_P2_AkumulacnyStoper.AlarmTime.IN:= TRUE;
				SC_P2_AkumulacnyStoper.Switch1:= TRUE;
			END_IF

			IF NOT P2_AkumulacnyStoper.IN.PritomnostPaletky THEN
				P2_AkumulacnyStoper.OUT.ZasunStoper:= FALSE;
				SC_P2_AkumulacnyStoper.ResetStep:= TRUE;
				SC_P2_AkumulacnyStoper.Step:= 100;
			ELSIF SC_P2_AkumulacnyStoper.AlarmTime.Q THEN
				P2_Alarmy[299]:= TRUE;
				P2_Pracovisko.STAV.Porucha_ST3:= TRUE;
			END_IF

			//*******************************************************Manuálny režim*******************************************************************************//
		700:
			SC_P2_AkumulacnyStoper.StepName:='700 - Manualny Rezim';
			SC_P2_AkumulacnyStoper.IdleTime.PT:= T#8s;
			SC_P2_AkumulacnyStoper.AlarmTime.PT:= T#5s;

	END_CASE

END_PROGRAM

PROGRAM _EXIT
	(* Insert code here *)

END_PROGRAM
```

#### Variables.var - Local variables
```iecst
VAR
	TEST : BOOL := 0;
END_VAR
```

### Program Logical/Program/Pracovisko_2/P2_StoperSrobovania (IEC)
